(* IEC 61131-3 sources: Industry-PLC-LLM/data/PLCBEAD_repo/PLCBEAD_PLCEmbed-main/PLC-BEAD/Source/OpenPLCv2 (part 7) *)

(* ---- MB_SERVER.ST ---- *)
TYPE
	oscat_IP_FIFO128_DATA  : ARRAY [1..128] OF BYTE;
	oscat_Mailbox  : ARRAY [1..16] OF BYTE;

	oscat_NW_BUF_SHORT : ARRAY [0..1407] OF BYTE;
	oscat_NW_BUF_LONG  : ARRAY [0..4095] OF BYTE;

	oscat_IP_FIFO_DATA :
	STRUCT
		X       : oscat_IP_FIFO128_DATA; (* IP_ID FIFO Speicher          *)
		Y       : oscat_IP_FIFO128_DATA; (* IP_ID Z�hler                 *)
		ID      : BYTE;                  (* h�chste vergabene id         *)
		MAX_ID  : BYTE;                  (* maximal Anmeldungen pro ID   *)
		INIT    : BOOL;                  (* Initialisierung durchgef�hrt *)
		EMPTY   : BOOL;                  (* FIFO leer                    *)
		FULL    : BOOL;                  (* FIFO voll                    *)
		TOP     : INT;                   (* maximale anzahl in FIFO      *)
		NW      : INT;                   (* Schreibzeiger                *)
		NR      : INT;                   (* Lesezeiger                   *)
	END_STRUCT;

	oscat_IP_C:
	STRUCT
		C_MODE:			BYTE;          		(*W Mode: TCP/UCP AKTIV/PASSIV                               *)
		C_PORT:         WORD;          		(*W Portnummer                                               *)
		C_IP:           DWORD;         		(*W IP-Adresse gepackt wwxxyyzz = www.xxx.yyy.zzz            *)
		C_STATE:        BYTE;          		(*R Verbindungsstatus ON/OFF + Flanke ON/OFF                 *)
		C_ENABLE:       BOOL;          		(*W Freigabe f�r Connect                                     *)
		R_OBSERVE:      BOOL;          		(*W Empfang ueberwachen                                      *)
		TIME_RESET:     BOOL;          		(*W Alle Timer ruecksetzen                                   *)
		ERROR:          DWORD;         		(*R vvwwxxyy (vv = CON_ERROR, ww = SEN_ERROR, xx = REC_ERROR *)
		FIFO:           oscat_IP_FIFO_DATA; (*I IP FIFO Struktur                                         *)
		MAILBOX:		oscat_Mailbox;		(*I Mailbox: Datenbereich f�r Bausteindatenaustausch         *)
	END_STRUCT;

	oscat_NETWORK_BUFFER :
	STRUCT
		SIZE   : UINT;
		BUFFER : oscat_NW_BUF_LONG;
	END_STRUCT;

	oscat_NETWORK_BUFFER_SHORT :
	STRUCT
	SIZE   : UINT;
	BUFFER : oscat_NW_BUF_SHORT;
	END_STRUCT;

	oscat_aW0_255	: ARRAY [0..255] OF WORD;
	oscat_VMAP_DATA :
	STRUCT
		FC       : DWORD;
		V_ADR    : INT;
		V_SIZE   : INT;
		P_ADR    : INT;
		TIME_OUT : TIME;
	END_STRUCT;

	oscat_MB_VMAP : ARRAY [1..10] OF oscat_VMAP_DATA;

	csv_parser_demo_col : ARRAY [1..4] OF REAL;
	csv_parser_demo     : ARRAY [1..2] OF csv_parser_demo_col;

END_TYPE

FUNCTION_BLOCK MB_VMAP_Block

	VAR_IN_OUT
		VMAP :	oscat_MB_VMAP;
	END_VAR

	VAR_INPUT
		FC :	INT;
		V_ADR :	INT;
		V_CNT :	INT;
		SIZE :	INT;
	END_VAR

	VAR_OUTPUT
		P_ADR :	INT;
		P_BIT :	INT;
		ERROR :	BYTE;
	END_VAR

	VAR
		i :	INT;
		vopt :	DWORD;
		vadr :	INT;
		padr :	INT;
		mask :	DWORD;
		vsize :	INT;
		w_tmp :	WORD;
		i_tmp :	INT;
		init :	BOOL;
	END_VAR

	IF init = FALSE THEN
		init := TRUE;
		IF VMAP[1].FC = DWORD#0 THEN
			VMAP[1].FC := DWORD#16#FFFF_FFFF;
			VMAP[1].V_ADR := 0;
			VMAP[1].V_SIZE := 256;
			VMAP[1].P_ADR := 0;
		END_IF;
	END_IF;

	ERROR := BYTE#02;
	mask := SHL(DWORD#1,FC);

	IF (mask AND DWORD#2#00000000_01000000_00000000_01100000) <> DWORD#0 THEN
		V_CNT := 1;
	ELSIF V_CNT = 0 THEN
		RETURN;
	END_IF;

	FOR i := 1 TO 10 DO
		vopt := VMAP[i].FC;
		IF (vopt AND mask) <> DWORD#0 THEN
			vadr := VMAP[i].V_ADR;
			vsize := VMAP[i].V_SIZE;
			padr := VMAP[i].P_ADR;

			IF (mask AND DWORD#2#00000000_00000000_10000000_00100110) <> DWORD#0 THEN
				i_tmp := WORD_TO_INT(SHR(INT_TO_WORD(V_ADR + V_CNT -1),4))+1;
				IF i_tmp <= SIZE AND i_tmp <= vsize THEN
					w_tmp := INT_TO_WORD(V_ADR);
					P_ADR := WORD_TO_INT(SHR(w_tmp,4)) + padr;
					P_BIT := WORD_TO_INT(w_tmp AND WORD#16#000F);
					ERROR := BYTE#0;
					EXIT;
				END_IF;
			ELSIF (mask AND DWORD#2#00000000_11000001_00000000_01011000) <> DWORD#0 THEN
				IF V_ADR >= vadr AND V_ADR + V_CNT <= vadr + vsize THEN
					P_ADR := V_ADR - vadr + padr;
					IF P_ADR + V_CNT <= SIZE THEN
						ERROR := BYTE#0;
						EXIT;
					END_IF;
				END_IF;
			ELSE
				ERROR := BYTE#01;
				RETURN;
			END_IF;
		END_IF;
	END_FOR;

	IF ERROR = BYTE#0 THEN
		IF (mask AND DWORD#2#00000000_11000001_10000000_01100000) <> DWORD#0 THEN
			VMAP[i].TIME_OUT := T#1ms;
		END_IF;
	END_IF;

END_FUNCTION_BLOCK

FUNCTION _BYTE_TO_INT:INT
	VAR_INPUT
		IN :	BYTE;
	END_VAR

	_BYTE_TO_INT := USINT_TO_INT(BYTE_TO_USINT(IN));
END_FUNCTION

FUNCTION_BLOCK IP_FIFO_Block

  VAR_IN_OUT
    FIFO :	oscat_IP_FIFO_DATA;
    ID :	BYTE;
    STATE :	BYTE;
  END_VAR

  VAR
    tmp :	INT;
  END_VAR

  IF NOT FIFO.INIT THEN
    FIFO.INIT		:= TRUE;
    FIFO.NW		:= 1;
    FIFO.NR		:= 1;
    FIFO.EMPTY	:= TRUE;
    FIFO.FULL		:= FALSE;
    FIFO.TOP		:= 128;
    FIFO.MAX_ID	:= BYTE#1;
  END_IF;

  IF ID = BYTE#00 THEN
    IF FIFO.ID < INT_TO_BYTE(FIFO.TOP) THEN
      ID := USINT_TO_BYTE(BYTE_TO_USINT(FIFO.ID) + USINT#1);
      FIFO.ID := ID ;

    ELSIF STATE < BYTE#200 THEN
      STATE := BYTE#255;
    RETURN;
    END_IF;
  END_IF;

  IF STATE = BYTE#1 AND NOT FIFO.FULL THEN
    tmp := _BYTE_TO_INT(ID);
    IF FIFO.Y[tmp] < FIFO.MAX_ID THEN
      FIFO.Y[tmp] := USINT_TO_BYTE(BYTE_TO_USINT(FIFO.Y[tmp]) + USINT#1);
      tmp := FIFO.NW;
      FIFO.X[tmp] := ID;
      IF FIFO.NW = FIFO.TOP THEN FIFO.NW := 1; ELSE FIFO.NW := FIFO.NW + 1; END_IF;
      FIFO.FULL := FIFO.NW = FIFO.NR;
    FIFO.EMPTY := FALSE;
      STATE := BYTE#2;
    END_IF;
  END_IF;

  IF STATE = BYTE#2 AND NOT FIFO.EMPTY THEN
    tmp := FIFO.NR;
    IF ID = FIFO.X[tmp] THEN
      STATE := BYTE#3;
    END_IF;
  END_IF;

  IF STATE = BYTE#4 AND NOT FIFO.EMPTY THEN

    tmp := FIFO.NR;
    IF ID = FIFO.X[tmp] THEN
      tmp := _BYTE_TO_INT(ID);
      FIFO.Y[tmp] := USINT_TO_BYTE(BYTE_TO_USINT(FIFO.Y[tmp]) - USINT#1);

      IF FIFO.NR = FIFO.TOP THEN FIFO.NR := 1; ELSE FIFO.NR := FIFO.NR + 1; END_IF;
      FIFO.EMPTY := FIFO.NR = FIFO.NW;
    FIFO.FULL := FALSE;
    END_IF;
    STATE := BYTE#5;
  END_IF;

END_FUNCTION_BLOCK

FUNCTION _UDINT_TO_TIME:TIME

	VAR_INPUT
		IN :	UDINT;
	END_VAR

	_UDINT_TO_TIME := DINT_TO_TIME(UDINT_TO_DINT(IN));

END_FUNCTION

FUNCTION_BLOCK T_PLC_MS_block

	VAR_OUTPUT
		T_PLC_MS :	UDINT;
	END_VAR

	VAR_EXTERNAL
		PLC_TICKS_PER_SEC :	INT;
		PLC_SYS_TICK_CNT :	DINT;
	END_VAR

	VAR
		debug :	BOOL;(*Debug-Mode ON / OFF*)
		N :	INT;(*Debug-Faktor*)
		Offset :	UDINT;(*Debug-Offset*)
		temp :	DWORD := DWORD#1;(*Debug-Offset*)
		mode :	BOOL;(*modus*)
		faktor :	UDINT;(*Systemtakt-Faktor*)
		init :	BOOL;
		v_plc_ticks_per_sec :	UDINT;
		base :	UDINT := UDINT#1000;
	END_VAR

	IF init = FALSE THEN
		v_plc_ticks_per_sec := INT_TO_UDINT(PLC_TICKS_PER_SEC);
		IF v_plc_ticks_per_sec = UDINT#1024 THEN
			faktor := UDINT#1;
			mode := FALSE;
		ELSIF v_plc_ticks_per_sec > UDINT#0 THEN
			IF v_plc_ticks_per_sec <= base THEN
				faktor := base / v_plc_ticks_per_sec;
				mode := FALSE;
			ELSE
				faktor := v_plc_ticks_per_sec / base;
				mode := TRUE;
			END_IF;
		ELSE
			faktor := UDINT#1;
		END_IF;
		init := TRUE;
	END_IF;

	IF mode THEN
		T_PLC_MS := DINT_TO_UDINT(PLC_SYS_TICK_CNT) / faktor;
	ELSE
		T_PLC_MS := DINT_TO_UDINT(PLC_SYS_TICK_CNT) * faktor;
	END_IF;

	IF debug THEN
		T_PLC_MS := (DWORD_TO_UDINT(SHL(UDINT_TO_DWORD(T_PLC_MS),N) OR SHL(temp,N)) - UDINT#1) + Offset;
	END_IF;

END_FUNCTION_BLOCK

FUNCTION WORD_OF_BYTE:WORD
	VAR_INPUT
		B1 :	BYTE;
		B0 :	BYTE;
	END_VAR
	WORD_OF_BYTE := SHL(BYTE_TO_WORD(B1),8) OR BYTE_TO_WORD(B0);
END_FUNCTION

FUNCTION BIT_LOAD_W:WORD
	VAR_INPUT
		IN :	WORD;
		VAL :	BOOL;
		POS :	INT;
	END_VAR

	IF VAL THEN
		BIT_LOAD_W := in OR SHL(WORD#1,pos);
	ELSE
		BIT_LOAD_W := in AND (NOT SHL(WORD#1,pos));
	END_IF;
END_FUNCTION

FUNCTION_BLOCK MB_SERVER_Block

	VAR_IN_OUT
		IP_C :	oscat_IP_C;
		S_BUF :	oscat_NETWORK_BUFFER_SHORT;
		R_BUF :	oscat_NETWORK_BUFFER_SHORT;
		VMAP :	oscat_MB_VMAP;
		DATA :	oscat_aW0_255;
	END_VAR

	VAR_INPUT
		DATA_SIZE :	INT;
		ENABLE :	BOOL;
		UDP :	BOOL;
	END_VAR

	VAR_OUTPUT
		ERROR :	DWORD;
	END_VAR

	VAR
		MB_VMAP :	MB_VMAP_Block;
		adr1 :	INT;
		adr2 :	INT;
		points :	INT;
		points2 :	INT;
		coils :	BYTE;
		mask :	BYTE;
		idx1 :	INT;
		idx2 :	INT;
		bit_pos :	INT;
		count :	INT;
		fc :	INT;
		i :	INT;
		state :	INT;
		IP_STATE :	BYTE;
		IP_ID :	BYTE;
		IP_FIFO :	IP_FIFO_Block;
		w_tmp :	WORD;
		last_cycle :	TIME;
		tx :	TIME;
		T_PLC_MS :	T_PLC_MS_Block;
		t :	TON;
		ip_error :	BOOL;
	END_VAR

	T_PLC_MS();
	tx := UDINT_TO_TIME(T_PLC_MS.T_PLC_MS);

	FOR i := 1 TO 10 DO
		IF VMAP[i].TIME_OUT > T#0s THEN
			VMAP[i].TIME_OUT := VMAP[i].TIME_OUT + tx - last_cycle;
		END_IF;
	END_FOR;
	last_cycle := tx;
	ip_error := IP_C.ERROR > DWORD#0;

	CASE state OF

	00:
		IF ENABLE THEN
			state := 10;
			IP_STATE := BYTE#1;
		END_IF;

	10:
		IF IP_STATE = BYTE#3 THEN

			IP_C.C_PORT     := WORD#0;
			IP_C.C_IP       := DWORD#0;
			IP_C.C_MODE     := SEL(UDP,BYTE#4,BYTE#5);
			IP_C.TIME_RESET := TRUE;
			IP_C.C_ENABLE   := TRUE;
			IP_C.R_OBSERVE  := FALSE;
			state := 20;
		END_IF;

	20:	IF NOT ip_error THEN
			IF S_BUF.SIZE = UINT#0 AND R_BUF.SIZE > UINT#6 THEN
				IF  R_BUF.SIZE = WORD_TO_UINT(WORD_OF_BYTE(R_BUF.BUFFER[4],R_BUF.BUFFER[5])) + UINT#6 THEN
					ERROR := DWORD#00;

					FOR i := 0 TO 13 DO
						S_BUF.BUFFER[i] := R_BUF.BUFFER[i];
					END_FOR;

					fc := _BYTE_TO_INT(R_BUF.BUFFER[7]);

					adr1 := WORD_TO_INT(WORD_OF_BYTE(R_BUF.BUFFER[8],R_BUF.BUFFER[9]));
					points := WORD_TO_INT(WORD_OF_BYTE(R_BUF.BUFFER[10],R_BUF.BUFFER[11]));

					MB_VMAP(VMAP:=VMAP,FC:=fc,V_ADR:=adr1,V_CNT:=points,SIZE:=DATA_SIZE);
					VMAP:=MB_VMAP.VMAP;
					adr1:=MB_VMAP.P_ADR;
					bit_pos:=MB_VMAP.P_BIT;
					ERROR:=BYTE_TO_DWORD(MB_VMAP.ERROR);

					IF ERROR = DWORD#0 THEN
						CASE fc OF

						1..2 :
							count := 9;
							coils := BYTE#0;
							mask := BYTE#1;
							FOR i := 1 TO points DO
								IF mask = BYTE#0 THEN
									mask := BYTE#1;
									S_BUF.BUFFER[count] := coils;
									coils := BYTE#0;
									count := count + 1;
								END_IF;
								IF (DATA[adr1] AND SHL(WORD#1,bit_pos)) > WORD#0 THEN
									coils := coils OR mask;
								END_IF;

								bit_Pos := bit_Pos + 1;
								IF bit_pos > 15 THEN
									adr1 := adr1 + 1;
									bit_pos := 0;
								END_IF;

								mask := SHL(mask,1);
							END_FOR;
							S_BUF.BUFFER[Count] := coils;

							S_BUF.BUFFER[8] := INT_TO_BYTE(count - 8);
							S_BUF.SIZE := INT_TO_UINT(count + 1);

						3..4 :
							idx1 := 07;
							count := adr1 + points - 1;
							FOR i := adr1 TO count DO
								idx1 := idx1 + 2;
								idx2 := idx1 + 1;
								w_tmp := DATA[i];
								S_BUF.BUFFER[idx1] := WORD_TO_BYTE(SHR(w_tmp,8));
								S_BUF.BUFFER[idx2] := WORD_TO_BYTE(w_tmp);
							END_FOR;
							S_BUF.BUFFER[8] := SHL(INT_TO_BYTE(points),1);
							S_BUF.SIZE := INT_TO_UINT(idx2 + 1);
						5 :
							DATA[adr1]:=BIT_LOAD_W(DATA[adr1],R_BUF.BUFFER[10]>BYTE#0,bit_pos);
							S_BUF.SIZE := UINT#12;
						6 :
							DATA[adr1] := WORD_OF_BYTE(R_BUF.BUFFER[10],R_BUF.BUFFER[11]);
							S_BUF.SIZE := UINT#12;
						15 :
							mask := BYTE#1;
							idx1 := 13;
							FOR i := 1 TO points DO
								DATA[adr1]:=BIT_LOAD_W(DATA[adr1],(R_BUF.BUFFER[idx1] AND mask)>BYTE#0,bit_pos);
								bit_pos := bit_pos + 1;
								IF bit_pos > 15 THEN
									adr1 := adr1 + 1;
									bit_pos := 0;
								END_IF;
								mask := ROL(mask,1);
								IF mask = BYTE#1 THEN
									idx1 := idx1 +1;
								END_IF;
							END_FOR;
							S_BUF.SIZE := UINT#12;
						16 :
							idx1 := 11;
							count := adr1 + points -1;
							FOR i := adr1 TO Count DO
								idx1 := idx1 + 2;
								idx2 := idx1 + 1;
								Data[i] := WORD_OF_BYTE(R_BUF.BUFFER[idx1],R_BUF.BUFFER[idx2]);
							END_FOR;
							S_BUF.SIZE := UINT#12;
						22 :
							w_tmp := WORD_OF_BYTE(R_BUF.BUFFER[11],R_BUF.BUFFER[11]);
							DATA[adr1] := (DATA[adr1] AND w_tmp) OR (WORD_OF_BYTE(R_BUF.BUFFER[12],R_BUF.BUFFER[13]) AND (NOT w_tmp));
							S_BUF.SIZE := UINT#14;
						23 :
							adr2 := WORD_TO_INT(WORD_OF_BYTE(R_BUF.BUFFER[12],R_BUF.BUFFER[13]));
							points2 := WORD_TO_INT(WORD_OF_BYTE(R_BUF.BUFFER[14],R_BUF.BUFFER[15]));

							MB_VMAP(VMAP:=VMAP,FC:=16,V_ADR:=adr2,V_CNT:=points2,SIZE:=DATA_SIZE);
							VMAP:=MB_VMAP.VMAP;
							adr2:=MB_VMAP.P_ADR;
							ERROR:=BYTE_TO_DWORD(MB_VMAP.ERROR);

							IF ERROR = DWORD#0 THEN
								idx1 := 15;
								count := adr2 + points2 -1;
								FOR i := adr2 TO count DO
									idx1 := idx1 + 2;
									idx2 := idx1 + 1;
									Data[i] := WORD_OF_BYTE(R_BUF.BUFFER[idx1],R_BUF.BUFFER[idx2]);
								END_FOR;

								idx1 := 07;
								count := adr1 + points - 1;
								FOR i := adr1 TO count DO
									idx1 := idx1 + 2;
									idx2 := idx1 + 1;
									w_tmp := DATA[i];
									S_BUF.BUFFER[idx1] := WORD_TO_BYTE(SHR(w_tmp,8));
									S_BUF.BUFFER[idx2] := WORD_TO_BYTE(w_tmp);
								END_FOR;
								S_BUF.BUFFER[8] := SHL(INT_TO_BYTE(points),1);
								S_BUF.SIZE := INT_TO_UINT(idx2 + 1);

							END_IF;

						ELSE
							ERROR := DWORD#01;
						END_CASE;
					END_IF;
				END_IF;

				IF ERROR > DWORD#0 THEN
					S_BUF.BUFFER[7] := S_BUF.BUFFER[7] OR BYTE#2#1000_0000;
					S_BUF.BUFFER[8] := DWORD_TO_BYTE(ERROR);
					S_BUF.SIZE := UINT#9;
				END_IF;

				S_BUF.BUFFER[4] := BYTE#0;
				S_BUF.BUFFER[5] := UINT_TO_BYTE(S_BUF.SIZE - UINT#6);

			END_IF;
		ELSE
			ERROR := IP_C.ERROR;
		END_IF;

		t(IN:= ip_error, PT:=T#5s);
		IF t.Q THEN
			IP_C.TIME_RESET := TRUE;
		END_IF;

		R_BUF.SIZE := UINT#0;

		IF ENABLE = FALSE THEN
			IP_STATE := BYTE#4;
			state := 00;
		END_IF;
	END_CASE;

	IP_FIFO(FIFO:=IP_C.FIFO,STATE:=IP_STATE,ID:=IP_ID);
	IP_C.FIFO:=IP_FIFO.FIFO;
	IP_STATE := IP_FIFO.STATE;
	IP_ID:=IP_FIFO.ID;

END_FUNCTION_BLOCK

PROGRAM program0
	VAR
		IP_C :	oscat_IP_C;
		S_BUF :	oscat_NETWORK_BUFFER_SHORT;
		R_BUF :	oscat_NETWORK_BUFFER_SHORT;
		VMAP :	oscat_MB_VMAP;
		DATA :	oscat_aW0_255;
		DATA_SIZE :	INT;
		ENABLE :	BOOL;
		UDP :	BOOL;
		ERROR :	DWORD;

		func_block : MB_SERVER_Block;
	END_VAR
	func_block.IP_C := IP_C;
	func_block.S_BUF := S_BUF;
	func_block.R_BUF := R_BUF;
	func_block.VMAP := VMAP;
	func_block.DATA := DATA;
	func_block.DATA_SIZE := DATA_SIZE;
	func_block.ENABLE := ENABLE;
	func_block.UDP := UDP;

	func_block();
  	IP_C  := func_block.IP_C;
	S_BUF  := func_block.S_BUF;
	R_BUF  := func_block.R_BUF;
	VMAP  := func_block.VMAP;
	DATA  := func_block.DATA;
	ERROR  := func_block.ERROR;

END_PROGRAM

CONFIGURATION Config0

	VAR_GLOBAL
		PLC_TICKS_PER_SEC :	INT;
		PLC_SYS_TICK_CNT :	DINT;
	END_VAR

  	RESOURCE Res0 ON PLC
    	TASK task0(INTERVAL := T#20ms,PRIORITY := 0);
    	PROGRAM instance0 WITH task0 : program0;
  	END_RESOURCE

END_CONFIGURATION

(* ---- MB_VMAP.ST ---- *)
TYPE
  oscat_VMAP_DATA :
  STRUCT
	FC       : DWORD;
    V_ADR    : INT;
    V_SIZE   : INT;
    P_ADR    : INT;
	TIME_OUT : TIME;
  END_STRUCT;

  oscat_MB_VMAP : ARRAY [1..10] OF oscat_VMAP_DATA;

  csv_parser_demo_col : ARRAY [1..4] OF REAL;
  csv_parser_demo     : ARRAY [1..2] OF csv_parser_demo_col;

END_TYPE

FUNCTION_BLOCK MB_VMAP_Block

	VAR_IN_OUT
		VMAP :	oscat_MB_VMAP;
	END_VAR

	VAR_INPUT
		FC :	INT;
		V_ADR :	INT;
		V_CNT :	INT;
		SIZE :	INT;
	END_VAR

	VAR_OUTPUT
		P_ADR :	INT;
		P_BIT :	INT;
		ERROR :	BYTE;
	END_VAR

	VAR
		i :	INT;
		vopt :	DWORD;
		vadr :	INT;
		padr :	INT;
		mask :	DWORD;
		vsize :	INT;
		w_tmp :	WORD;
		i_tmp :	INT;
		init :	BOOL;
	END_VAR

	IF init = FALSE THEN
		init := TRUE;
		IF VMAP[1].FC = DWORD#0 THEN
			VMAP[1].FC := DWORD#16#FFFF_FFFF;
			VMAP[1].V_ADR := 0;
			VMAP[1].V_SIZE := 256;
			VMAP[1].P_ADR := 0;
		END_IF;
	END_IF;

	ERROR := BYTE#02;
	mask := SHL(DWORD#1,FC);

	IF (mask AND DWORD#2#00000000_01000000_00000000_01100000) <> DWORD#0 THEN
		V_CNT := 1;
	ELSIF V_CNT = 0 THEN
		RETURN;
	END_IF;

	FOR i := 1 TO 10 DO
		vopt := VMAP[i].FC;
		IF (vopt AND mask) <> DWORD#0 THEN
			vadr := VMAP[i].V_ADR;
			vsize := VMAP[i].V_SIZE;
			padr := VMAP[i].P_ADR;

			IF (mask AND DWORD#2#00000000_00000000_10000000_00100110) <> DWORD#0 THEN
				i_tmp := WORD_TO_INT(SHR(INT_TO_WORD(V_ADR + V_CNT -1),4))+1;
				IF i_tmp <= SIZE AND i_tmp <= vsize THEN
					w_tmp := INT_TO_WORD(V_ADR);
					P_ADR := WORD_TO_INT(SHR(w_tmp,4)) + padr;
					P_BIT := WORD_TO_INT(w_tmp AND WORD#16#000F);
					ERROR := BYTE#0;
					EXIT;
				END_IF;
			ELSIF (mask AND DWORD#2#00000000_11000001_00000000_01011000) <> DWORD#0 THEN
				IF V_ADR >= vadr AND V_ADR + V_CNT <= vadr + vsize THEN
					P_ADR := V_ADR - vadr + padr;
					IF P_ADR + V_CNT <= SIZE THEN
						ERROR := BYTE#0;
						EXIT;
					END_IF;
				END_IF;
			ELSE
				ERROR := BYTE#01;
				RETURN;
			END_IF;
		END_IF;
	END_FOR;

	IF ERROR = BYTE#0 THEN
		IF (mask AND DWORD#2#00000000_11000001_10000000_01100000) <> DWORD#0 THEN
			VMAP[i].TIME_OUT := T#1ms;
		END_IF;
	END_IF;

END_FUNCTION_BLOCK

PROGRAM program0
	VAR
		VMAP :	oscat_MB_VMAP;
		FC :	INT;
		V_ADR :	INT;
		V_CNT :	INT;
		SIZE :	INT;
		P_ADR :	INT;
		P_BIT :	INT;
		ERROR :	BYTE;

		func_block : MB_VMAP_Block;
	END_VAR
	func_block.VMAP := VMAP;
	func_block.V_ADR := V_ADR;
	func_block.FC := FC;
	func_block.V_CNT := V_CNT;
	func_block.SIZE := SIZE;

	func_block();
  	VMAP  := func_block.VMAP;
	P_ADR  := func_block.P_ADR;
	P_BIT  := func_block.P_BIT;
	ERROR  := func_block.ERROR;
END_PROGRAM

CONFIGURATION Config0
	RESOURCE Res0 ON PLC
		TASK task0(INTERVAL := T#20ms,PRIORITY := 0);
		PROGRAM instance0 WITH task0 : program0;
	END_RESOURCE
END_CONFIGURATION

(* ---- MESSAGE_4R.ST ---- *)
FUNCTION INC1:INT

	VAR_INPUT
		X :	INT;
		N :	INT;
	END_VAR

	IF X >= N - 1 THEN
		INC1 := 0;
	ELSE
		INC1 := X + 1;
	END_IF;
END_FUNCTION

FUNCTION_BLOCK MESSAGE_4R_Block

	VAR_INPUT
		M0 :	STRING;
		M1 :	STRING;
		M2 :	STRING;
		M3 :	STRING;
		MM :	INT := 3;
		ENQ :	BOOL := TRUE;
		CLK :	BOOL := TRUE;
		T1 :	TIME := T#3s;
	END_VAR

	VAR_OUTPUT
		MX :	STRING;
		MN :	INT;
		TR :	BOOL;
	END_VAR

	VAR
		timer :	TON;
		edge :	BOOL;
	END_VAR

	TR := FALSE;
	IF ENQ THEN
		IF (NOT edge AND clk) OR timer.q THEN
				MN := INC1(MN, MM);
				TR := TRUE;
				timer(in := FALSE);
				CASE MN OF
					0 : MX := M0;
					1 : MX := M1;
					2 : MX := M2;
					3 : MX := M3;
				END_CASE;
		END_IF;
		edge := clk;
		timer( in := CLK, pt := T1);
	ELSE
		MX := '';
		MN := 0;
	END_IF;

END_FUNCTION_BLOCK

PROGRAM program0

	VAR
		M0 :	STRING;
		M1 :	STRING;
		M2 :	STRING;
		M3 :	STRING;
		MM :	INT;
		ENQ :	BOOL;
		CLK :	BOOL;
		T1 :	TIME;

		MX :	STRING;
		MN :	INT;
		TR :	BOOL;

		func_block : MESSAGE_4R_Block;
	END_VAR

	func_block.M0 := M0;
	func_block.M1 := M1;
	func_block.M2 := M2;
	func_block.M3 := M3;
	func_block.MM := MM;
	func_block.ENQ := ENQ;
	func_block.CLK := CLK;
	func_block.T1 := T1;

	func_block();

	MX := func_block.MX;
	MN := func_block.MN;
	TR := func_block.TR;

END_PROGRAM

CONFIGURATION Config0

	RESOURCE Res0 ON PLC
		TASK task0(INTERVAL := T#20ms,PRIORITY := 0);
		PROGRAM instance0 WITH task0 : program0;
	END_RESOURCE

END_CONFIGURATION

(* ---- MESSAGE_8.ST ---- *)
FUNCTION_BLOCK MESSAGE_8_Block

	VAR_INPUT
		IN1 :	BOOL;
		IN2 :	BOOL;
		IN3 :	BOOL;
		IN4 :	BOOL;
		IN5 :	BOOL;
		IN6 :	BOOL;
		IN7 :	BOOL;
		IN8 :	BOOL;
		S1 :	STRING;
		S2 :	STRING;
		S3 :	STRING;
		S4 :	STRING;
		S5 :	STRING;
		S6 :	STRING;
		S7 :	STRING;
		S8 :	STRING;
	END_VAR

	VAR_OUTPUT
		M :	STRING;
	END_VAR

	IF in1 THEN
		M := S1;
	ELSIF in2 THEN
		M := S2;
	ELSIF in3 THEN
		M := S3;
	ELSIF in4 THEN
		M := S4;
	ELSIF in5 THEN
		M := S5;
	ELSIF in6 THEN
		M := S6;
	ELSIF in7 THEN
		M := S7;
	ELSIF in8 THEN
		M := S8;
	ELSE
		M := '';
	END_IF;

END_FUNCTION_BLOCK

PROGRAM program0

	VAR
		IN1 :	BOOL;
		IN2 :	BOOL;
		IN3 :	BOOL;
		IN4 :	BOOL;
		IN5 :	BOOL;
		IN6 :	BOOL;
		IN7 :	BOOL;
		IN8 :	BOOL;
		S1 :	STRING;
		S2 :	STRING;
		S3 :	STRING;
		S4 :	STRING;
		S5 :	STRING;
		S6 :	STRING;
		S7 :	STRING;
		S8 :	STRING;

		M :	STRING;

		func_block : MESSAGE_8_Block;
	END_VAR

	func_block.IN1 := IN1;
	func_block.IN2 := IN2;
	func_block.IN3 := IN3;
	func_block.IN4 := IN4;
	func_block.IN5 := IN5;
	func_block.IN6 := IN6;
	func_block.IN7 := IN7;
	func_block.IN8 := IN8;
	func_block.S1 := S1;
	func_block.S2 := S2;
	func_block.S3 := S3;
	func_block.S4 := S4;
	func_block.S5 := S5;
	func_block.S6 := S6;
	func_block.S7 := S7;
	func_block.S8 := S8;

	func_block();

	M  := func_block.M;

END_PROGRAM

CONFIGURATION Config0

	VAR_GLOBAL
		PLC_TICKS_PER_SEC :	INT;
		PLC_SYS_TICK_CNT :	DINT;
	END_VAR

	RESOURCE Res0 ON PLC
		TASK task0(INTERVAL := T#20ms,PRIORITY := 0);
		PROGRAM instance0 WITH task0 : program0;
	END_RESOURCE

END_CONFIGURATION

(* ---- METER.ST ---- *)
TYPE REAL2:

	STRUCT
		R1 : REAL;
		RX : REAL;
	END_STRUCT;

END_TYPE

FUNCTION_BLOCK R2_ADD_Block

	VAR_INPUT
		X :	REAL2;
		Y :	REAL;
	END_VAR

	VAR_OUTPUT
		R2_ADD :	REAL2;
	END_VAR

	VAR
		temp :	REAL;
	END_VAR

	temp := X.RX;
	R2_ADD.RX := Y + X.R1 + X.RX;
	R2_ADD.R1 := temp - R2_ADD.RX + Y + X.R1;

END_FUNCTION_BLOCK

FUNCTION_BLOCK T_PLC_MS_Block
	VAR_OUTPUT
		T_PLC_MS :	UDINT;
	END_VAR

	VAR_EXTERNAL
		PLC_TICKS_PER_SEC :	INT;
		PLC_SYS_TICK_CNT :	DINT;
	END_VAR

	VAR
		debug :	BOOL;(*Debug-Mode ON / OFF*)
		N :	INT;(*Debug-Faktor*)
		Offset :	UDINT;(*Debug-Offset*)
		temp :	DWORD := DWORD#1;(*Debug-Offset*)
		mode :	BOOL;(*modus*)
		faktor :	UDINT;(*Systemtakt-Faktor*)
		init :	BOOL;
		v_plc_ticks_per_sec :	UDINT;
		base :	UDINT := UDINT#1000;
	END_VAR

	IF init = FALSE THEN
		v_plc_ticks_per_sec := INT_TO_UDINT(PLC_TICKS_PER_SEC);
		IF v_plc_ticks_per_sec = UDINT#1024 THEN
			faktor := UDINT#1;
			mode := FALSE;
		ELSIF v_plc_ticks_per_sec > UDINT#0 THEN
			IF v_plc_ticks_per_sec <= base THEN
				faktor := base / v_plc_ticks_per_sec;
				mode := FALSE;
			ELSE
				faktor := v_plc_ticks_per_sec / base;
				mode := TRUE;
			END_IF;
		ELSE
			faktor := UDINT#1;
		END_IF;
		init := TRUE;
	END_IF;

	IF mode THEN
		T_PLC_MS := DINT_TO_UDINT(PLC_SYS_TICK_CNT) / faktor;
	ELSE
		T_PLC_MS := DINT_TO_UDINT(PLC_SYS_TICK_CNT) * faktor;
	END_IF;

	IF debug THEN
		T_PLC_MS := (DWORD_TO_UDINT(SHL(UDINT_TO_DWORD(T_PLC_MS),N) OR SHL(temp,N)) - UDINT#1) + Offset;
	END_IF;
END_FUNCTION_BLOCK

FUNCTION_BLOCK METER_Block

	VAR_INPUT
		M1 :	REAL;
		M2 :	REAL;
		I1 :	BOOL;
		I2 :	BOOL;
		D :	REAL := 1.0;
		RST :	BOOL;
	END_VAR

	VAR_IN_OUT
		MX :	REAL;
	END_VAR

	VAR RETAIN
		MR :	REAL2;
	END_VAR

	VAR
		MX1 :	REAL;(*current consumption value on M1 and M2*)
		MX2 :	REAL;(*current consumption value on M1 and M2*)
		tx :	UDINT;
		last :	UDINT;
		tc :	REAL;
		init :	BOOL;
		T_PLC_MS :	T_PLC_MS_Block;
		R2_ADD :	R2_ADD_Block;
	END_VAR

	T_PLC_MS();
	tx:= T_PLC_MS.T_PLC_MS;
	IF NOT init THEN
		init := TRUE;
		last := tx;
		mr.RX := mx;
		mr.R1 := 0.0;
	ELSIF tx = last THEN
		RETURN;
	ELSE
		tc := UDINT_TO_REAL(tx - last) * 0.001;
	END_IF;
	last := tx;

	(* reset *)
	IF rst THEN
		mr.R1 := 0.0;
		mr.RX := 0.0;
	ELSE
		MX1 := SEL(I1,0.0,M1);
		MX2 := SEL(I2,0.0,M2);
		R2_ADD(X:=MR,Y:=(SEL(I1,0.0,mx1) + SEL(I2, 0.0, mx2)) / D * TC);
		MR:=R2_ADD.R2_ADD;
		MX := mr.RX;
	END_IF;

END_FUNCTION_BLOCK

PROGRAM program0

	VAR
		M1 :	REAL;
		M2 :	REAL;
		I1 :	BOOL;
		I2 :	BOOL;
		D :	REAL := 1.0;
		RST :	BOOL;

		MX :	REAL;

		func_block : METER_Block;
	END_VAR

	func_block.M1 := M1;
	func_block.M2 := M2;
	func_block.I1 := I1;
	func_block.I2 := I2;
	func_block.D := D;
	func_block.RST := RST;
	func_block.MX := MX;

	func_block();

	MX  := func_block.MX;

END_PROGRAM

CONFIGURATION Config0

	VAR_GLOBAL
		PLC_TICKS_PER_SEC :	INT;
		PLC_SYS_TICK_CNT :	DINT;
	END_VAR

	RESOURCE Res0 ON PLC
		TASK task0(INTERVAL := T#20ms,PRIORITY := 0);
		PROGRAM instance0 WITH task0 : program0;
	END_RESOURCE

END_CONFIGURATION

(* ---- METER_STAT.ST ---- *)
FUNCTION DAY_OF_WEEK:INT

	VAR_INPUT
		IDATE :	UDINT;
	END_VAR

	DAY_OF_WEEK := UDINT_TO_INT((idate / UDINT#86400 + UDINT#3) MOD UDINT#7) + INT#01;
END_FUNCTION

FUNCTION LEAP_OF_DATE:BOOL

	VAR_INPUT
		IDATE :	UDINT;
	END_VAR

	LEAP_OF_DATE := SHL(UDINT_TO_DWORD((idate + UDINT#43200) / UDINT#31557600), 30) = DWORD#16#80000000;
END_FUNCTION

FUNCTION DAY_OF_YEAR:INT
	VAR_INPUT
		IDATE :	UDINT;
	END_VAR

	DAY_OF_YEAR := UDINT_TO_INT(((idate) / UDINT#86400) MOD UDINT#1461);
	IF DAY_OF_YEAR > 729 THEN
		IF DAY_OF_YEAR > 1095 THEN DAY_OF_YEAR := DAY_OF_YEAR - 1095; ELSE DAY_OF_YEAR := DAY_OF_YEAR - 729; END_IF;
	ELSIF DAY_OF_YEAR > 364 THEN
		DAY_OF_YEAR := DAY_OF_YEAR - 364;
	ELSE
		DAY_OF_YEAR := DAY_OF_YEAR + 1;
	END_IF;
END_FUNCTION

FUNCTION MONTH_OF_DATE:INT

	VAR_INPUT
		IDATE :	UDINT;
	END_VAR

	MONTH_OF_DATE := DAY_OF_YEAR(idate);
	IF MONTH_OF_DATE < 32 THEN
		MONTH_OF_DATE := 1;
	ELSIF LEAP_OF_DATE((IDATE)) THEN
		MONTH_OF_DATE := (MONTH_OF_DATE * 53 + 1668) / 1623;
	ELSE
		MONTH_OF_DATE := (MONTH_OF_DATE * 53 + 1700) / 1620;
	END_IF;
END_FUNCTION

FUNCTION YEAR_OF_DATE:INT
	VAR_INPUT
		IDATE :	UDINT;
	END_VAR

	YEAR_OF_DATE := UDINT_TO_INT((idate+UDINT#43200) / UDINT#31557600 + UDINT#1970);
END_FUNCTION

FUNCTION_BLOCK METER_STAT_Block

	VAR_INPUT
		IN :	REAL;
		DI :	UDINT;
		RST :	BOOL;
	END_VAR

	VAR_IN_OUT
		LAST_DAY :	REAL;
		CURRENT_DAY :	REAL;
		LAST_WEEK :	REAL;
		CURRENT_WEEK :	REAL;
		LAST_MONTH :	REAL;
		CURRENT_MONTH :	REAL;
		LAST_YEAR :	REAL;
		CURRENT_YEAR :	REAL;
	END_VAR

	VAR RETAIN
		year_start :	REAL;
		month_start :	REAL;
		week_start :	REAL;
		day_start :	REAL;
		last_run :	UDINT;
	END_VAR

	IF rst THEN
		Last_Day := 0.0;
		Current_Day := 0.0;
		Day_start := IN;
		Last_week := 0.0;
		Current_week := 0.0;
		Week_start := in;
		Last_month := 0.0;
		Current_month := 0.0;
		month_start := in;
		last_year := 0.0;
		current_year := 0.0;
		year_start := in;
	ELSE
		Current_Day := IN - Day_Start;
		Current_Week := In - Week_Start;
		Current_Month := IN - Month_Start;
		Current_Year := IN - Year_Start;
	END_IF;

	IF YEAR_OF_DATE(DI) > YEAR_OF_DATE(last_run) THEN
		(* a new year has started *)
		last_year := current_year;
		current_year := 0.0;
		year_start := in;
		last_month := current_month;
		current_month := 0.0;
		month_start := in;
		last_day := current_day;
		current_day := 0.0;
		day_start := in;
	ELSIF MONTH_OF_DATE(DI) > MONTH_OF_DATE(last_run) THEN
		(* a new month has started, january is alrerady done by year change *)
		last_month := current_month;
		current_month := 0.0;
		month_start := in;
		last_day := current_day;
		current_day := 0.0;
		day_start := in;
	ELSIF DAY_OF_YEAR(di) > DAY_OF_YEAR(last_run) THEN
		(* day has chaged, first day of year and first day of month has already been taken care of *)
		last_day := current_day;
		current_day := 0.0;
		day_start := in;
	END_IF;
	IF DAY_OF_WEEK(DI) < DAY_OF_WEEK(last_run) THEN
		(* a new week has started *)
		last_week := current_week;
		current_week := 0.0;
		week_start := in;
	END_IF;
	last_run := di;

END_FUNCTION_BLOCK

PROGRAM program0

	VAR
		IN :	REAL;
		DI :	UDINT;
		RST :	BOOL;

		LAST_DAY :	REAL;
		CURRENT_DAY :	REAL;
		LAST_WEEK :	REAL;
		CURRENT_WEEK :	REAL;
		LAST_MONTH :	REAL;
		CURRENT_MONTH :	REAL;
		LAST_YEAR :	REAL;
		CURRENT_YEAR :	REAL;

		func_block : METER_STAT_Block;
	END_VAR

	func_block.IN := IN;
	func_block.DI := DI;
	func_block.RST := RST;
	func_block.LAST_DAY := LAST_DAY;
	func_block.CURRENT_DAY := CURRENT_DAY;
	func_block.LAST_WEEK := LAST_WEEK;
	func_block.CURRENT_WEEK := CURRENT_WEEK;
	func_block.LAST_MONTH := LAST_MONTH;
	func_block.CURRENT_MONTH := CURRENT_MONTH;
	func_block.LAST_YEAR := LAST_YEAR;
	func_block.CURRENT_YEAR := CURRENT_YEAR;

	func_block();

	LAST_DAY  := func_block.LAST_DAY;
	CURRENT_DAY  := func_block.CURRENT_DAY;
	LAST_WEEK  := func_block.LAST_WEEK;
	CURRENT_WEEK  := func_block.CURRENT_WEEK;
	LAST_MONTH  := func_block.LAST_MONTH;
	CURRENT_MONTH  := func_block.CURRENT_MONTH;
	LAST_YEAR  := func_block.LAST_YEAR;
	CURRENT_YEAR  := func_block.CURRENT_YEAR;

END_PROGRAM

CONFIGURATION Config0

	VAR_GLOBAL
		PLC_TICKS_PER_SEC :	INT;
		PLC_SYS_TICK_CNT :	DINT;
	END_VAR

	RESOURCE Res0 ON PLC
		TASK task0(INTERVAL := T#20ms,PRIORITY := 0);
		PROGRAM instance0 WITH task0 : program0;
	END_RESOURCE

END_CONFIGURATION

(* ---- MIRROR.ST ---- *)
FUNCTION_BLOCK MIRROR_Block

	VAR_INPUT
		STR :	STRING;
	END_VAR

	VAR_OUTPUT
		MIRROR :	STRING;
	END_VAR

	VAR
		i :	INT;
		st_temp :	STRING;
	END_VAR

	mirror := '';
	i := LEN(str);
	WHILE i > 0 DO
	st_temp := MID(str,1,i);
	mirror := CONCAT(mirror,st_temp);
	i := i -1;
	END_WHILE;

END_FUNCTION_BLOCK

PROGRAM program0

	VAR
		STR :	STRING;
		MIRROR :	STRING;
		func_block : MIRROR_Block;
	END_VAR
	func_block.STR := STR;
	func_block();
	MIRROR  := func_block.MIRROR;

END_PROGRAM

CONFIGURATION Config0

	RESOURCE Res0 ON PLC
		TASK task0(INTERVAL := T#20ms,PRIORITY := 0);
		PROGRAM instance0 WITH task0 : program0;
	END_RESOURCE

END_CONFIGURATION

(* ---- MONTH_TO_STRING.ST ---- *)
TYPE
  oscat_ELEMENT_MONTHS 	: ARRAY [1..12] OF STRING;
  oscat_MONTHS			: ARRAY [1..3]  OF oscat_ELEMENT_MONTHS := [0, 0, 0];
  oscat_ELEMENT_MONTHS3	: ARRAY [1..12] OF STRING;
  oscat_MONTHS3			: ARRAY [1..3]  OF oscat_ELEMENT_MONTHS3 := [0,0,0];
END_TYPE

TYPE oscat_LANGUAGE:
  STRUCT
    DEFAULT 	: INT;
	LMAX    	: INT;
  END_STRUCT;
END_TYPE

FUNCTION_BLOCK SETUP_LANGUAGE_Block

	VAR_IN_OUT
		LANGUAGE :	oscat_LANGUAGE;
	END_VAR

	VAR
		init :	BOOL;
	END_VAR

	IF init THEN RETURN; END_IF;
	init := TRUE;

	LANGUAGE.DEFAULT  := 1; (* 1=english, 2=german 3=french *)
	LANGUAGE.LMAX := 3;
END_FUNCTION_BLOCK

FUNCTION_BLOCK SETUP_MONTHS3_Block

	VAR_IN_OUT
		MONTHS3 :	oscat_MONTHS3;
	END_VAR

	VAR
		init :	BOOL;
	END_VAR

	IF init THEN RETURN; END_IF;
	init := TRUE;

	(* ---- english --- *)
	MONTHS3[1][01] := 'Jan';
	MONTHS3[1][02] := 'Feb';
	MONTHS3[1][03] := 'Mar';
	MONTHS3[1][04] := 'Apr';
	MONTHS3[1][05] := 'May';
	MONTHS3[1][06] := 'Jun';
	MONTHS3[1][07] := 'Jul';
	MONTHS3[1][08] := 'Aug';
	MONTHS3[1][09] := 'Sep';
	MONTHS3[1][10] := 'Oct';
	MONTHS3[1][11] := 'Nov';
	MONTHS3[1][12] := 'Dec';

	(* ---- german --- *)
	MONTHS3[2][01] := 'Jan';
	MONTHS3[2][02] := 'Feb';
	MONTHS3[2][03] := 'Mrz';
	MONTHS3[2][04] := 'Apr';
	MONTHs3[2][05] := 'Mai';
	MONTHS3[2][06] := 'Jun';
	MONTHS3[2][07] := 'Jul';
	MONTHS3[2][08] := 'Aug';
	MONTHS3[2][09] := 'Sep';
	MONTHS3[2][10] := 'Okt';
	MONTHS3[2][11] := 'Nov';
	MONTHS3[2][12] := 'Dez';

	(* ---- french --- *)
	MONTHS3[3][01] := 'Jan';
	MONTHS3[3][02] := 'Fev';
	MONTHS3[3][03] := 'Mar';
	MONTHS3[3][04] := 'Avr';
	MONTHs3[3][05] := 'Mai';
	MONTHS3[3][06] := 'Jun';
	MONTHS3[3][07] := 'Jul';
	MONTHS3[3][08] := 'Aou';
	MONTHS3[3][09] := 'Sep';
	MONTHS3[3][10] := 'Oct';
	MONTHS3[3][11] := 'Nov';
	MONTHS3[3][12] := 'Dec';
	(*@KEY@: END_WORKSHEET *)
END_FUNCTION_BLOCK

FUNCTION_BLOCK SETUP_MONTHS_Block

	VAR_IN_OUT
		MONTHS :	oscat_MONTHS;
	END_VAR

	VAR
		init :	BOOL;
	END_VAR

	IF init THEN RETURN; END_IF;
	init := TRUE;

	(* ---- english --- *)
	MONTHS[1][01] := 'January';
	MONTHS[1][02] := 'February';
	MONTHS[1][03] := 'March';
	MONTHS[1][04] := 'April';
	MONTHS[1][05] := 'May';
	MONTHS[1][06] := 'June';
	MONTHS[1][07] := 'July';
	MONTHS[1][08] := 'August';
	MONTHS[1][09] := 'September';
	MONTHS[1][10] := 'October';
	MONTHS[1][11] := 'November';
	MONTHS[1][12] := 'December';

	(* ---- german --- *)
	MONTHS[2][01] := 'Januar';
	MONTHS[2][02] := 'Februar';
	MONTHS[2][03] := 'March';
	MONTHS[2][04] := 'April';
	MONTHS[2][05] := 'Mai';
	MONTHS[2][06] := 'Juni';
	MONTHS[2][07] := 'Juli';
	MONTHS[2][08] := 'August';
	MONTHS[2][09] := 'September';
	MONTHS[2][10] := 'Oktober';
	MONTHS[2][11] := 'November';
	MONTHS[2][12] := 'Dezember';

	(* ---- french --- *)
	MONTHS[3][01] := 'Janvier';
	MONTHS[3][02] := 'Fvrier';
	MONTHS[3][03] := 'mars';
	MONTHS[3][04] := 'Avril';
	MONTHS[3][05] := 'Mai';
	MONTHS[3][06] := 'Juin';
	MONTHS[3][07] := 'Juillet';
	MONTHS[3][08] := 'Aot';
	MONTHS[3][09] := 'Septembre';
	MONTHS[3][10] := 'Octobre';
	MONTHS[3][11] := 'Novembre';
	MONTHS[3][12] := 'Decembre';
END_FUNCTION_BLOCK

FUNCTION_BLOCK MONTH_TO_STRING_Block

	VAR_INPUT
		MTH :	INT;
		LANG :	INT;
		LX :	INT;
	END_VAR

	VAR_OUTPUT
		MONTH_TO_STRING :	STRING;
	END_VAR

	VAR
		LY :	INT;
		SETUP_MONTHS :	SETUP_MONTHS_Block;
		MONTHS :	oscat_MONTHS;
		SETUP_MONTHS3 :	SETUP_MONTHS3_Block;
		MONTHS3 :	oscat_MONTHS3;
		SETUP_LANGUAGE :	SETUP_LANGUAGE_Block;
		LANGUAGE :	oscat_LANGUAGE;
	END_VAR

	SETUP_MONTHS(MONTHS:=MONTHS);
	MONTHS:=SETUP_MONTHS.MONTHS;
	SETUP_MONTHS3(MONTHS3:=MONTHS3);
	MONTHS3:=SETUP_MONTHS3.MONTHS3;
	SETUP_LANGUAGE(LANGUAGE:=LANGUAGE);
	LANGUAGE:=SETUP_LANGUAGE.LANGUAGE;

	IF LANG = 0 THEN Ly := LANGUAGE.DEFAULT; ELSE ly := MIN(LANG, language.LMAX); END_IF;
	IF MTH < 1 OR MTH > 12 THEN
		RETURN;
	ELSIF LX = 0 THEN
		MONTH_TO_STRING := MONTHS[ly][MTH];
	ELSIF Lx = 3 THEN
		MONTH_TO_STRING := MONTHS3[ly][MTH];
	END_IF;

END_FUNCTION_BLOCK

PROGRAM program0
	VAR
		MTH :	INT;
		LANG :	INT;
		LX :	INT;
		MONTH_TO_STRING :	STRING;
		func_block : MONTH_TO_STRING_Block;
	END_VAR
		func_block.MTH  := MTH;
		func_block.LANG  := LANG;
		func_block.LX  := LX;
		func_block();
		MONTH_TO_STRING := func_block.MONTH_TO_STRING;
END_PROGRAM

CONFIGURATION Config0
	RESOURCE Res0 ON PLC
		TASK task0(INTERVAL := T#20ms,PRIORITY := 0);
		PROGRAM instance0 WITH task0 : program0;
	END_RESOURCE
END_CONFIGURATION

(* ---- MOON_PHASE.ST ---- *)
FUNCTION TIME_TO_UDINT2:UDINT
	VAR_INPUT
		X :	TIME;
	END_VAR

	TIME_TO_UDINT2 := DINT_TO_UDINT(TIME_TO_DINT(X));
END_FUNCTION

FUNCTION_BLOCK MOON_PHASE_Block

	VAR_INPUT
		XDT :	UDINT;
		SCALE :	BYTE := BYTE#12;
		UPDATE :	TIME := T#1h;
	END_VAR

	VAR_OUTPUT
		PHASE :	BYTE;
	END_VAR

	VAR
		x :	UDINT;
		last_dt :	UDINT;
	END_VAR

	IF XDT - last_dt > TIME_TO_UDINT2(UPDATE) THEN
		x := (XDT - UDINT#603240) MOD UDINT#2551392;
		PHASE := UDINT_TO_BYTE(BYTE_TO_UDINT(SCALE) * x / UDINT#2551392) ;
		last_dt := XDT;
	END_IF;

END_FUNCTION_BLOCK

PROGRAM program0
	VAR
		XDT :	UDINT;
		SCALE :	BYTE := BYTE#12;
		UPDATE :	TIME := T#1h;
		PHASE :	BYTE;

		func_block : MOON_PHASE_Block;
	END_VAR
	func_block.XDT := XDT;
	func_block.SCALE := SCALE;
	func_block.UPDATE := UPDATE;

	func_block();
  	PHASE  := func_block.PHASE;
END_PROGRAM

CONFIGURATION Config0
	RESOURCE Res0 ON PLC
		TASK task0(INTERVAL := T#20ms,PRIORITY := 0);
		PROGRAM instance0 WITH task0 : program0;
	END_RESOURCE
END_CONFIGURATION

(* ---- NET_VAR_BOOL8.ST ---- *)
TYPE

	oscat_NW_BUF_LONG  : ARRAY [0..4095] OF BYTE;

	oscat_NETWORK_BUFFER :
	STRUCT
		SIZE   : UINT;
		BUFFER : oscat_NW_BUF_LONG;
	END_STRUCT;

END_TYPE

TYPE oscat_NET_VAR_DATA :
	STRUCT
		CYCLE : UDINT;
		STATE : BYTE;
		INDEX : INT;
		ID_MAX : USINT;
		ERROR_ID : BYTE;
		BUF_SIZE : UINT;
		S_BUF : oscat_NETWORK_BUFFER;
		R_BUF : oscat_NETWORK_BUFFER;
	END_STRUCT;
END_TYPE

FUNCTION BIT_OF_DWORD : BOOL
  VAR_INPUT
    IN : DWORD;
    N : INT;
  END_VAR

  BIT_OF_DWORD := (SHR(in,N) AND 16#00000001) > 0;
END_FUNCTION

FUNCTION_BLOCK BYTE_TO_BITS_Block
	VAR_INPUT
		IN :	BYTE;
	END_VAR

	VAR_OUTPUT
		B0 :	BOOL;
		B1 :	BOOL;
		B2 :	BOOL;
		B3 :	BOOL;
		B4 :	BOOL;
		B5 :	BOOL;
		B6 :	BOOL;
		B7 :	BOOL;
	END_VAR

	B0 := BIT_OF_DWORD(BYTE_TO_DWORD(IN),0); (* IN.X0 *)
	B1 := BIT_OF_DWORD(BYTE_TO_DWORD(IN),1); (* IN.X1 *)
	B2 := BIT_OF_DWORD(BYTE_TO_DWORD(IN),2); (* IN.X2 *)
	B3 := BIT_OF_DWORD(BYTE_TO_DWORD(IN),3); (* IN.X3 *)
	B4 := BIT_OF_DWORD(BYTE_TO_DWORD(IN),4); (* IN.X4 *)
	B5 := BIT_OF_DWORD(BYTE_TO_DWORD(IN),5); (* IN.X5 *)
	B6 := BIT_OF_DWORD(BYTE_TO_DWORD(IN),6); (* IN.X6 *)
	B7 := BIT_OF_DWORD(BYTE_TO_DWORD(IN),7); (* IN.X7 *)
END_FUNCTION_BLOCK

FUNCTION BYTE_OF_BIT:BYTE
	VAR_INPUT
		B0 :	BOOL;
		B1 :	BOOL;
		B2 :	BOOL;
		B3 :	BOOL;
		B4 :	BOOL;
		B5 :	BOOL;
		B6 :	BOOL;
		B7 :	BOOL;
	END_VAR
	Byte_of_bit := SHL(SHL(SHL(SHL(SHL(SHL(SHL(BOOL_TO_BYTE(B7),1) OR BOOL_TO_BYTE(B6),1)
	OR BOOL_TO_BYTE(B5),1) OR BOOL_TO_BYTE(B4),1) OR BOOL_TO_BYTE(B3),1) OR BOOL_TO_BYTE(B2),1)
	OR BOOL_TO_BYTE(B1),1) OR BOOL_TO_BYTE(B0);
END_FUNCTION

FUNCTION_BLOCK NET_VAR_BOOL8_Block

	VAR_INPUT
		IN1 :	BOOL;
		IN2 :	BOOL;
		IN3 :	BOOL;
		IN4 :	BOOL;
		IN5 :	BOOL;
		IN6 :	BOOL;
		IN7 :	BOOL;
		IN8 :	BOOL;
	END_VAR

	VAR_OUTPUT
		OUT1 :	BOOL;
		OUT2 :	BOOL;
		OUT3 :	BOOL;
		OUT4 :	BOOL;
		OUT5 :	BOOL;
		OUT6 :	BOOL;
		OUT7 :	BOOL;
		OUT8 :	BOOL;
		ID :	BYTE;
	END_VAR

	VAR_IN_OUT
		X :	oscat_NET_VAR_DATA;
	END_VAR

	VAR
		init :	BOOL;
		index :	INT;
		index2 :	INT;
		_BYTE_TO_BITS :	BYTE_TO_BITS_Block;
	END_VAR

	IF NOT init THEN
		init := TRUE;
		X.ID_MAX := X.ID_MAX + USINT#1;
		ID := USINT_TO_BYTE(X.ID_MAX);
	END_IF;

	IF X.STATE > BYTE#0 AND X.ERROR_ID = BYTE#0 THEN
		index := X.index;
		IF INT_TO_UINT(index + 3) > X.BUF_SIZE THEN
			X.ERROR_ID := ID;
		ELSE
			IF X.STATE = BYTE#1 THEN
				X.S_BUF.BUFFER[index] := ID;
				index := index + 1;
				X.S_BUF.BUFFER[index] := BYTE#4;
				index := index + 1;
				X.S_BUF.BUFFER[index] := BYTE_OF_BIT(IN1,IN2,IN3,IN4,IN5,IN6,IN7,IN8);
				index := index + 1;

			ELSIF X.STATE = BYTE#2 THEN
				index2 := index + 1;
				IF X.R_BUF.BUFFER[index] <> ID OR X.R_BUF.BUFFER[index2] <> BYTE#4 THEN
					X.ERROR_ID := ID;
				ELSE
					index := index + 2;
					_BYTE_TO_BITS(IN:=X.R_BUF.BUFFER[index]);
					OUT1 := _BYTE_TO_BITS.B0;
					OUT2 := _BYTE_TO_BITS.B1;
					OUT3 := _BYTE_TO_BITS.B2;
					OUT4 := _BYTE_TO_BITS.B3;
					OUT5 := _BYTE_TO_BITS.B4;
					OUT6 := _BYTE_TO_BITS.B5;
					OUT7 := _BYTE_TO_BITS.B6;
					OUT8 := _BYTE_TO_BITS.B7;
					index := index + 1;
				END_IF;
			END_IF;
			X.index := index;
		END_IF;
	END_IF;

END_FUNCTION_BLOCK

PROGRAM program0
	VAR
		IN1 :	BOOL;
		IN2 :	BOOL;
		IN3 :	BOOL;
		IN4 :	BOOL;
		IN5 :	BOOL;
		IN6 :	BOOL;
		IN7 :	BOOL;
		IN8 :	BOOL;
		OUT1 :	BOOL;
		OUT2 :	BOOL;
		OUT3 :	BOOL;
		OUT4 :	BOOL;
		OUT5 :	BOOL;
		OUT6 :	BOOL;
		OUT7 :	BOOL;
		OUT8 :	BOOL;
		ID :	BYTE;
		X :	oscat_NET_VAR_DATA;

		func_block : NET_VAR_BOOL8_Block;
	END_VAR
	func_block.IN1 := IN1;
	func_block.IN2 := IN2;
	func_block.IN3 := IN3;
	func_block.IN4 := IN4;
	func_block.IN5 := IN5;
	func_block.IN6 := IN6;
	func_block.IN7 := IN7;
	func_block.IN8 := IN8;
	func_block.X := X;

	func_block();
  	OUT1  := func_block.OUT1;
	OUT2  := func_block.OUT2;
	OUT3  := func_block.OUT3;
	OUT4  := func_block.OUT4;
	OUT5  := func_block.OUT5;
	OUT6  := func_block.OUT6;
	OUT7  := func_block.OUT7;
	OUT8  := func_block.OUT8;
	ID  := func_block.ID;
	X  := func_block.X;
END_PROGRAM

CONFIGURATION Config0
	RESOURCE Res0 ON PLC
		TASK task0(INTERVAL := T#20ms,PRIORITY := 0);
		PROGRAM instance0 WITH task0 : program0;
	END_RESOURCE
END_CONFIGURATION

(* ---- NET_VAR_BUFFER.ST ---- *)
TYPE
	oscat_aB1_64 : ARRAY[1..64] OF BYTE;
END_TYPE

TYPE

	oscat_NW_BUF_LONG  : ARRAY [0..4095] OF BYTE;

	oscat_NETWORK_BUFFER :
	STRUCT
		SIZE   : UINT;
		BUFFER : oscat_NW_BUF_LONG;
	END_STRUCT;

END_TYPE

TYPE oscat_NET_VAR_DATA :
	STRUCT
		CYCLE : UDINT;
		STATE : BYTE;
		INDEX : INT;
		ID_MAX : USINT;
		ERROR_ID : BYTE;
		BUF_SIZE : UINT;
		S_BUF : oscat_NETWORK_BUFFER;
		R_BUF : oscat_NETWORK_BUFFER;
	END_STRUCT;
END_TYPE

FUNCTION_BLOCK NET_VAR_BUFFER_Block

	VAR_OUTPUT
		ID :	BYTE;
	END_VAR

	VAR_IN_OUT
		BUF_IN :	oscat_aB1_64;
		BUF_OUT :	oscat_aB1_64;
		X :	oscat_NET_VAR_DATA;
	END_VAR

	VAR
		size :	INT;
		init :	BOOL;
		index :	INT;
		index2 :	INT;
	END_VAR

	IF NOT init THEN
		init := TRUE;
		X.ID_MAX := X.ID_MAX + USINT#1;
		ID := USINT_TO_BYTE(X.ID_MAX);
	END_IF;

	IF X.STATE > BYTE#0 AND X.ERROR_ID = BYTE#0 THEN
		index := X.index;
		IF X.STATE = BYTE#1 THEN
			size := 64;
			IF INT_TO_UINT(index + 3 + size) > X.BUF_SIZE THEN
				X.ERROR_ID := ID;
			ELSE
				X.S_BUF.BUFFER[index] := ID;
				index := index + 1;
				X.S_BUF.BUFFER[index] := BYTE#20;
				index := index + 1;
				X.S_BUF.BUFFER[index] := INT_TO_BYTE(size);
				index := index + 1;
				FOR index2 := 1 TO size DO
					X.S_BUF.BUFFER[index] := BUF_IN[index2];
					index := index + 1;
				END_FOR;
			END_IF;
		ELSIF X.STATE = BYTE#2 THEN
			index2 := index + 1;
			IF X.R_BUF.BUFFER[index] <> ID OR X.R_BUF.BUFFER[index2] <> BYTE#20 THEN
				X.ERROR_ID := ID;
			ELSE
				index := index + 2;
				size := BYTE_TO_INT(X.R_BUF.BUFFER[index]);
				index := index + 1;
				FOR index2 := 1 TO size DO
					BUF_OUT[index2] := X.R_BUF.BUFFER[index];
					index := index + 1;
				END_FOR;
			END_IF;
		END_IF;
		X.index := index;
	END_IF;

END_FUNCTION_BLOCK

PROGRAM program0
	VAR
		BUF_IN :	oscat_aB1_64;
		BUF_OUT :	oscat_aB1_64;
		X :	oscat_NET_VAR_DATA;
		ID :	BYTE;

		func_block : NET_VAR_BUFFER_Block;
	END_VAR
	func_block.BUF_IN := BUF_IN;
	func_block.BUF_OUT := BUF_OUT;
	func_block.X := X;

	func_block();
  	BUF_IN  := func_block.BUF_IN;
	BUF_OUT  := func_block.BUF_OUT;
	X  := func_block.X;
	ID  := func_block.ID;

END_PROGRAM

CONFIGURATION Config0
	RESOURCE Res0 ON PLC
		TASK task0(INTERVAL := T#20ms,PRIORITY := 0);
		PROGRAM instance0 WITH task0 : program0;
	END_RESOURCE
END_CONFIGURATION

(* ---- NET_VAR_DWORD8.ST ---- *)
TYPE
	oscat_nv_dw : ARRAY[1..8] OF DWORD;
END_TYPE

TYPE

	oscat_NW_BUF_LONG  : ARRAY [0..4095] OF BYTE;

	oscat_NETWORK_BUFFER :
	STRUCT
		SIZE   : UINT;
		BUFFER : oscat_NW_BUF_LONG;
	END_STRUCT;

END_TYPE

TYPE oscat_NET_VAR_DATA :
	STRUCT
		CYCLE : UDINT;
		STATE : BYTE;
		INDEX : INT;
		ID_MAX : USINT;
		ERROR_ID : BYTE;
		BUF_SIZE : UINT;
		S_BUF : oscat_NETWORK_BUFFER;
		R_BUF : oscat_NETWORK_BUFFER;
	END_STRUCT;
END_TYPE

FUNCTION_BLOCK NET_VAR_DWORD8_Block

	VAR_INPUT
		IN1 :	DWORD;
		IN2 :	DWORD;
		IN3 :	DWORD;
		IN4 :	DWORD;
		IN5 :	DWORD;
		IN6 :	DWORD;
		IN7 :	DWORD;
		IN8 :	DWORD;
	END_VAR

	VAR_OUTPUT
		OUT1 :	DWORD;
		OUT2 :	DWORD;
		OUT3 :	DWORD;
		OUT4 :	DWORD;
		OUT5 :	DWORD;
		OUT6 :	DWORD;
		OUT7 :	DWORD;
		OUT8 :	DWORD;
		ID :	BYTE;
	END_VAR

	VAR_IN_OUT
		X :	oscat_NET_VAR_DATA;
	END_VAR

	VAR
		init :	BOOL;
		i :	INT;
		i2 :	INT;
		index :	INT;
		index2 :	INT;
		ra :	oscat_nv_dw;
	END_VAR

	IF NOT init THEN
		init := TRUE;
		X.ID_MAX := X.ID_MAX + USINT#1;
		ID := USINT_TO_BYTE(X.ID_MAX);
	END_IF;

	IF X.STATE > BYTE#0 AND X.ERROR_ID = BYTE#0 THEN
		index := X.index;
		IF INT_TO_UINT(index + 34) > X.BUF_SIZE THEN
			X.ERROR_ID := ID;
		ELSE
			IF X.STATE = BYTE#1 THEN
				ra[1] := IN1;
				ra[2] := IN2;
				ra[3] := IN3;
				ra[4] := IN4;
				ra[5] := IN5;
				ra[6] := IN6;
				ra[7] := IN7;
				ra[8] := IN8;
				X.S_BUF.BUFFER[index] := ID;
				index := index + 1;
				X.S_BUF.BUFFER[index] := BYTE#13;
				index := index + 1;
				FOR i2 := 1 TO 8 DO
					FOR i := 1 TO 4 DO
						X.S_BUF.BUFFER[index] := DWORD_TO_BYTE(ra[i2]);
						ra[i2] := ROR(ra[i2],8);
						index := index + 1;
					END_FOR;
				END_FOR;

			ELSIF X.STATE = BYTE#2 THEN
				index2 := index + 1;
				IF X.R_BUF.BUFFER[index] <> ID OR X.R_BUF.BUFFER[index2] <> BYTE#13 THEN
					X.ERROR_ID := ID;
				ELSE
					index := index + 2;
					FOR i2 := 1 TO 8 DO
						ra[i2] := DWORD#0;
						FOR i := 1 TO 4 DO
							ra[i2] := ra[i2] OR BYTE_TO_DWORD(X.R_BUF.BUFFER[index]);
							ra[i2] := ROR(ra[i2],8);
							index := index + 1;
						END_FOR;
					END_FOR;
					OUT1 := ra[1];
					OUT2 := ra[2];
					OUT3 := ra[3];
					OUT4 := ra[4];
					OUT5 := ra[5];
					OUT6 := ra[6];
					OUT7 := ra[7];
					OUT8 := ra[8];
				END_IF;
			END_IF;
			X.index := index;
		END_IF;
	END_IF;

END_FUNCTION_BLOCK

PROGRAM program0
	VAR
		IN1 :	DWORD;
		IN2 :	DWORD;
		IN3 :	DWORD;
		IN4 :	DWORD;
		IN5 :	DWORD;
		IN6 :	DWORD;
		IN7 :	DWORD;
		IN8 :	DWORD;
		OUT1 :	DWORD;
		OUT2 :	DWORD;
		OUT3 :	DWORD;
		OUT4 :	DWORD;
		OUT5 :	DWORD;
		OUT6 :	DWORD;
		OUT7 :	DWORD;
		OUT8 :	DWORD;
		ID :	BYTE;
		X :	oscat_NET_VAR_DATA;

		func_block : NET_VAR_DWORD8_Block;
	END_VAR
	func_block.IN1 := IN1;
	func_block.IN2 := IN2;
	func_block.IN3 := IN3;
	func_block.IN4 := IN4;
	func_block.IN5 := IN5;
	func_block.IN6 := IN6;
	func_block.IN7 := IN7;
	func_block.IN8 := IN8;
	func_block.X := X;

	func_block();
  	OUT1  := func_block.OUT1;
	OUT2  := func_block.OUT2;
	OUT3  := func_block.OUT3;
	OUT4  := func_block.OUT4;
	OUT5  := func_block.OUT5;
	OUT6  := func_block.OUT6;
	OUT7  := func_block.OUT7;
	OUT8  := func_block.OUT8;
	ID  := func_block.ID;
	X  := func_block.X;
END_PROGRAM

CONFIGURATION Config0
	RESOURCE Res0 ON PLC
		TASK task0(INTERVAL := T#20ms,PRIORITY := 0);
		PROGRAM instance0 WITH task0 : program0;
	END_RESOURCE
END_CONFIGURATION

(* ---- ONTIME.ST ---- *)
FUNCTION_BLOCK T_PLC_MS_block
	VAR_OUTPUT
		T_PLC_MS :	UDINT;
	END_VAR

	VAR_EXTERNAL
		PLC_TICKS_PER_SEC :	INT;
		PLC_SYS_TICK_CNT :	DINT;
	END_VAR

	VAR
		debug :	BOOL;(*Debug-Mode ON / OFF*)
		N :	INT;(*Debug-Faktor*)
		Offset :	UDINT;(*Debug-Offset*)
		temp :	DWORD := DWORD#1;(*Debug-Offset*)
		mode :	BOOL;(*modus*)
		faktor :	UDINT;(*Systemtakt-Faktor*)
		init :	BOOL;
		v_plc_ticks_per_sec :	UDINT;
		base :	UDINT := UDINT#1000;
	END_VAR

	IF init = FALSE THEN
		v_plc_ticks_per_sec := INT_TO_UDINT(PLC_TICKS_PER_SEC);
		IF v_plc_ticks_per_sec = UDINT#1024 THEN
			faktor := UDINT#1;
			mode := FALSE;
		ELSIF v_plc_ticks_per_sec > UDINT#0 THEN
			IF v_plc_ticks_per_sec <= base THEN
				faktor := base / v_plc_ticks_per_sec;
				mode := FALSE;
			ELSE
				faktor := v_plc_ticks_per_sec / base;
				mode := TRUE;
			END_IF;
		ELSE
			faktor := UDINT#1;
		END_IF;
		init := TRUE;
	END_IF;

	IF mode THEN
		T_PLC_MS := DINT_TO_UDINT(PLC_SYS_TICK_CNT) / faktor;
	ELSE
		T_PLC_MS := DINT_TO_UDINT(PLC_SYS_TICK_CNT) * faktor;
	END_IF;

	IF debug THEN
		T_PLC_MS := (DWORD_TO_UDINT(SHL(UDINT_TO_DWORD(T_PLC_MS),N) OR SHL(temp,N)) - UDINT#1) + Offset;
	END_IF;

END_FUNCTION_BLOCK

FUNCTION_BLOCK ONTIME_Block

	VAR_INPUT
		IN :	BOOL;
		RST :	BOOL;
	END_VAR

	VAR_IN_OUT
		SECONDS :	UDINT;
		CYCLES :	UDINT;
	END_VAR

	VAR
		tx :	UDINT;
		last :	UDINT;
		edge :	BOOL;
		init :	BOOL;
		ms :	UDINT;
		T_PLC_MS :	T_PLC_MS_Block;
	END_VAR

	T_PLC_MS();
	tx:= T_PLC_MS.T_PLC_MS;

	IF NOT init THEN
		init := TRUE;
		last := tx;
		ms := UDINT#0;
	END_IF;
	IF RST THEN
		SECONDS := UDINT#0;
		CYCLES := UDINT#0;
		last := tx;
		ms := UDINT#0;
	ELSIF IN THEN
		(* add the current milliseconds *)
		ms := (tx - last) + ms;
		IF ms >= UDINT#1000 THEN
			seconds := seconds + UDINT#1;
			ms := ms - UDINT#1000;
		END_IF;
		cycles := cycles + BOOL_TO_UDINT(NOT edge);
	END_IF;
	last := tx;
	edge := in;

END_FUNCTION_BLOCK

PROGRAM program0
	VAR
		IN :	BOOL;
		RST :	BOOL;
		SECONDS :	UDINT;
		CYCLES :	UDINT;
		func_block : ONTIME_Block;
	END_VAR
	func_block.IN := IN;
	func_block.RST := RST;
	func_block();
	SECONDS  := func_block.SECONDS;
	CYCLES  := func_block.CYCLES;
END_PROGRAM

CONFIGURATION Config0
	VAR_GLOBAL
		PLC_TICKS_PER_SEC :	INT;
		PLC_SYS_TICK_CNT :	DINT;
	END_VAR
  	RESOURCE Res0 ON PLC
    	TASK task0(INTERVAL := T#20ms,PRIORITY := 0);
    	PROGRAM instance0 WITH task0 : program0;
  	END_RESOURCE
END_CONFIGURATION

(* ---- PARSET.ST ---- *)
TYPE
	oscat_parset_X              : ARRAY [1..4]    OF REAL;
	oscat_parset                : ARRAY [0..3]    OF oscat_parset_X := [0,0,0,0];
END_TYPE

FUNCTION TIME_TO_UDINT2:UDINT
	VAR_INPUT
		X :	TIME;
	END_VAR

	TIME_TO_UDINT2 := DINT_TO_UDINT(TIME_TO_DINT(X));
END_FUNCTION

FUNCTION _BYTE_TO_INT:INT
	VAR_INPUT
		IN :	BYTE;
	END_VAR

	_BYTE_TO_INT := USINT_TO_INT(BYTE_TO_USINT(IN));
END_FUNCTION

FUNCTION BIT_OF_DWORD : BOOL
  VAR_INPUT
    IN : DWORD;
    N : INT;
  END_VAR

  BIT_OF_DWORD := (SHR(in,N) AND 16#00000001) > 0;
  (* from OSCAT library; www.oscat.de  *)
END_FUNCTION

FUNCTION BIT_LOAD_B:BYTE
	VAR_INPUT
		IN :	BYTE;
		VAL :	BOOL;
		POS :	INT;
	END_VAR

	IF VAL THEN
		BIT_LOAD_B := in OR SHL(BYTE#1,pos);
	ELSE
		BIT_LOAD_B := in AND (NOT SHL(BYTE#1,pos));
	END_IF;
END_FUNCTION

FUNCTION_BLOCK T_PLC_MS_block
	VAR_OUTPUT
		T_PLC_MS :	UDINT;
	END_VAR

	VAR_EXTERNAL
		PLC_TICKS_PER_SEC :	INT;
		PLC_SYS_TICK_CNT :	DINT;
	END_VAR

	VAR
		debug :	BOOL;(*Debug-Mode ON / OFF*)
		N :	INT;(*Debug-Faktor*)
		Offset :	UDINT;(*Debug-Offset*)
		temp :	DWORD := DWORD#1;(*Debug-Offset*)
		mode :	BOOL;(*modus*)
		faktor :	UDINT;(*Systemtakt-Faktor*)
		init :	BOOL;
		v_plc_ticks_per_sec :	UDINT;
		base :	UDINT := UDINT#1000;
	END_VAR

	IF init = FALSE THEN
		v_plc_ticks_per_sec := INT_TO_UDINT(PLC_TICKS_PER_SEC);
		IF v_plc_ticks_per_sec = UDINT#1024 THEN
			faktor := UDINT#1;
			mode := FALSE;
		ELSIF v_plc_ticks_per_sec > UDINT#0 THEN
			IF v_plc_ticks_per_sec <= base THEN
				faktor := base / v_plc_ticks_per_sec;
				mode := FALSE;
			ELSE
				faktor := v_plc_ticks_per_sec / base;
				mode := TRUE;
			END_IF;
		ELSE
			faktor := UDINT#1;
		END_IF;
		init := TRUE;
	END_IF;

	IF mode THEN
		T_PLC_MS := DINT_TO_UDINT(PLC_SYS_TICK_CNT) / faktor;
	ELSE
		T_PLC_MS := DINT_TO_UDINT(PLC_SYS_TICK_CNT) * faktor;
	END_IF;

	IF debug THEN
		T_PLC_MS := (DWORD_TO_UDINT(SHL(UDINT_TO_DWORD(T_PLC_MS),N) OR SHL(temp,N)) - UDINT#1) + Offset;
	END_IF;
END_FUNCTION_BLOCK

FUNCTION_BLOCK PARSET_Block

	VAR_INPUT
		A0 :	BOOL;
		A1 :	BOOL;
		X01 :	REAL;
		X02 :	REAL;
		X03 :	REAL;
		X04 :	REAL;
		X11 :	REAL;
		X12 :	REAL;
		X13 :	REAL;
		X14 :	REAL;
		X21 :	REAL;
		X22 :	REAL;
		X23 :	REAL;
		X24 :	REAL;
		X31 :	REAL;
		X32 :	REAL;
		X33 :	REAL;
		X34 :	REAL;
		TC :	TIME;
	END_VAR

	VAR_OUTPUT
		P1 :	REAL;
		P2 :	REAL;
		P3 :	REAL;
		P4 :	REAL;
	END_VAR

	VAR
		X :	oscat_parset;
		S1 :	REAL;
		S2 :	REAL;
		S3 :	REAL;
		S4 :	REAL;
		tx :	UDINT;
		last :	UDINT;
		start :	BOOL;
		set :	BYTE;
		set2 :	INT;
		init :	BOOL;
		T_PLC_MS :	T_PLC_MS_Block;
	END_VAR

	(*@KEY@: WORKSHEET
	NAME: PARSET
	IEC_LANGUAGE: ST
	*)
	(* read system_time *)
	T_PLC_MS();
	tx:= T_PLC_MS.T_PLC_MS;

	(* init sequence *)
	IF NOT init THEN
		set:=BIT_LOAD_B(set,NOT A0,0); (* set.X0 := NOT A0; *)
		init := TRUE;
		X[0][1] := X01;
		X[0][2] := X02;
		X[0][3] := X03;
		X[0][4] := X04;
		X[1][1] := X11;
		X[1][2] := X12;
		X[1][3] := X13;
		X[1][4] := X14;
		X[2][1] := X21;
		X[2][2] := X22;
		X[2][3] := X23;
		X[2][4] := X24;
		X[3][1] := X31;
		X[3][2] := X32;
		X[3][3] := X33;
		X[3][4] := X34;
		P1 := X01;
		P2 := X02;
		P3 := X03;
		P4 := X04;
	END_IF;

	(* check for input change *)
	IF (A0 XOR BIT_OF_DWORD(BYTE_TO_DWORD(set),0)) OR (A1 XOR BIT_OF_DWORD(BYTE_TO_DWORD(set),1)) THEN  (* set.X0  ,  set.X1 *)
		(* a new set is selected *)
		set := BIT_LOAD_B(set,A0,0); (* set.X0 := A0; *)
		set := BIT_LOAD_B(set,A1,1); (* set.X1 := A1; *)

		IF tc > t#0s THEN
			start := TRUE;
			last := tx;
			(* save the step speed for the output changes in S *)
			set2 := _BYTE_TO_INT(set);
			S1 := (X[set2][1] - P1)/TIME_TO_REAL(tc);
			S2 := (X[set2][2] - P2)/TIME_TO_REAL(tc);
			S3 := (X[set2][3] - P3)/TIME_TO_REAL(tc);
			S4 := (X[set2][4] - P4)/TIME_TO_REAL(tc);
		END_IF;
	ELSIF start AND tx - last < TIME_TO_UDINT2(tc) THEN
		(* ramp the outputs to the new value *)
		set2 := _BYTE_TO_INT(set);
		P1 := X[set2][1] - S1*(TIME_TO_REAL(Tc) - UDINT_TO_REAL(tx + last));
		P2 := X[set2][2] - S2*(TIME_TO_REAL(Tc) - UDINT_TO_REAL(tx + last));
		P3 := X[set2][3] - S3*(TIME_TO_REAL(Tc) - UDINT_TO_REAL(tx + last));
		P4 := X[set2][4] - S4*(TIME_TO_REAL(Tc) - UDINT_TO_REAL(tx + last));
	ELSE
		(* make sure outputs match the correct set values *)
		set2 := _BYTE_TO_INT(set);
		start := FALSE;
		P1 := X[set2][1];
		P2 := X[set2][2];
		P3 := X[set2][3];
		P4 := X[set2][4];
	END_IF;

END_FUNCTION_BLOCK

PROGRAM program0

	VAR
		A0 :	BOOL;
		A1 :	BOOL;
		X01 :	REAL;
		X02 :	REAL;
		X03 :	REAL;
		X04 :	REAL;
		X11 :	REAL;
		X12 :	REAL;
		X13 :	REAL;
		X14 :	REAL;
		X21 :	REAL;
		X22 :	REAL;
		X23 :	REAL;
		X24 :	REAL;
		X31 :	REAL;
		X32 :	REAL;
		X33 :	REAL;
		X34 :	REAL;
		TC :	TIME;

		P1 :	REAL;
		P2 :	REAL;
		P3 :	REAL;
		P4 :	REAL;
		func_block : PARSET_Block;
  	END_VAR
	func_block.A0 := A0;
	func_block.A1 := A1;
	func_block.X01 := X01;
	func_block.X02 := X02;
	func_block.X03 := X03;
	func_block.X04 := X04;
	func_block.X11 := X11;
	func_block.X12 := X12;
	func_block.X13 := X13;
	func_block.X14 := X14;
	func_block.X21 := X21;
	func_block.X22 := X22;
	func_block.X23 := X23;
	func_block.X24 := X24;
	func_block.X31 := X31;
	func_block.X32 := X32;
	func_block.X33 := X33;
	func_block.X34 := X34;
	func_block.TC := TC;
	func_block();
	P1 := func_block.P1;
	P2 := func_block.P2;
	P3 := func_block.P3;
	P4 := func_block.P4;

END_PROGRAM

CONFIGURATION Config0

	VAR_GLOBAL
		PLC_TICKS_PER_SEC :	INT;
		PLC_SYS_TICK_CNT :	DINT;
	END_VAR

  	RESOURCE Res0 ON PLC
    	TASK task0(INTERVAL := T#20ms,PRIORITY := 0);
    	PROGRAM instance0 WITH task0 : program0;
  	END_RESOURCE

END_CONFIGURATION

(* ---- PARSET2.ST ---- *)
TYPE
	oscat_parset_X              : ARRAY [1..4]    OF REAL;
	oscat_parset                : ARRAY [0..3]    OF oscat_parset_X := [0,0,0,0];
END_TYPE

FUNCTION TIME_TO_UDINT2:UDINT
	VAR_INPUT
		X :	TIME;
	END_VAR

	TIME_TO_UDINT2 := DINT_TO_UDINT(TIME_TO_DINT(X));
END_FUNCTION

FUNCTION _BYTE_TO_INT:INT
	VAR_INPUT
		IN :	BYTE;
	END_VAR

	_BYTE_TO_INT := USINT_TO_INT(BYTE_TO_USINT(IN));
END_FUNCTION

FUNCTION BIT_OF_DWORD : BOOL
  VAR_INPUT
    IN : DWORD;
    N : INT;
  END_VAR

  BIT_OF_DWORD := (SHR(in,N) AND 16#00000001) > 0;
  (* from OSCAT library; www.oscat.de  *)
END_FUNCTION

FUNCTION BIT_LOAD_B:BYTE
	VAR_INPUT
		IN :	BYTE;
		VAL :	BOOL;
		POS :	INT;
	END_VAR

	IF VAL THEN
		BIT_LOAD_B := in OR SHL(BYTE#1,pos);
	ELSE
		BIT_LOAD_B := in AND (NOT SHL(BYTE#1,pos));
	END_IF;
END_FUNCTION

FUNCTION_BLOCK T_PLC_MS_block
	VAR_OUTPUT
		T_PLC_MS :	UDINT;
	END_VAR

	VAR_EXTERNAL
		PLC_TICKS_PER_SEC :	INT;
		PLC_SYS_TICK_CNT :	DINT;
	END_VAR

	VAR
		debug :	BOOL;(*Debug-Mode ON / OFF*)
		N :	INT;(*Debug-Faktor*)
		Offset :	UDINT;(*Debug-Offset*)
		temp :	DWORD := DWORD#1;(*Debug-Offset*)
		mode :	BOOL;(*modus*)
		faktor :	UDINT;(*Systemtakt-Faktor*)
		init :	BOOL;
		v_plc_ticks_per_sec :	UDINT;
		base :	UDINT := UDINT#1000;
	END_VAR

	IF init = FALSE THEN
		v_plc_ticks_per_sec := INT_TO_UDINT(PLC_TICKS_PER_SEC);
		IF v_plc_ticks_per_sec = UDINT#1024 THEN
			faktor := UDINT#1;
			mode := FALSE;
		ELSIF v_plc_ticks_per_sec > UDINT#0 THEN
			IF v_plc_ticks_per_sec <= base THEN
				faktor := base / v_plc_ticks_per_sec;
				mode := FALSE;
			ELSE
				faktor := v_plc_ticks_per_sec / base;
				mode := TRUE;
			END_IF;
		ELSE
			faktor := UDINT#1;
		END_IF;
		init := TRUE;
	END_IF;

	IF mode THEN
		T_PLC_MS := DINT_TO_UDINT(PLC_SYS_TICK_CNT) / faktor;
	ELSE
		T_PLC_MS := DINT_TO_UDINT(PLC_SYS_TICK_CNT) * faktor;
	END_IF;

	IF debug THEN
		T_PLC_MS := (DWORD_TO_UDINT(SHL(UDINT_TO_DWORD(T_PLC_MS),N) OR SHL(temp,N)) - UDINT#1) + Offset;
	END_IF;
END_FUNCTION_BLOCK

FUNCTION_BLOCK PARSET_Block

	VAR_INPUT
		A0 :	BOOL;
		A1 :	BOOL;
		X01 :	REAL;
		X02 :	REAL;
		X03 :	REAL;
		X04 :	REAL;
		X11 :	REAL;
		X12 :	REAL;
		X13 :	REAL;
		X14 :	REAL;
		X21 :	REAL;
		X22 :	REAL;
		X23 :	REAL;
		X24 :	REAL;
		X31 :	REAL;
		X32 :	REAL;
		X33 :	REAL;
		X34 :	REAL;
		TC :	TIME;
	END_VAR

	VAR_OUTPUT
		P1 :	REAL;
		P2 :	REAL;
		P3 :	REAL;
		P4 :	REAL;
	END_VAR

	VAR
		X :	oscat_parset;
		S1 :	REAL;
		S2 :	REAL;
		S3 :	REAL;
		S4 :	REAL;
		tx :	UDINT;
		last :	UDINT;
		start :	BOOL;
		set :	BYTE;
		set2 :	INT;
		init :	BOOL;
		T_PLC_MS :	T_PLC_MS_Block;
	END_VAR

	(*@KEY@: WORKSHEET
	NAME: PARSET
	IEC_LANGUAGE: ST
	*)
	(* read system_time *)
	T_PLC_MS();
	tx:= T_PLC_MS.T_PLC_MS;

	(* init sequence *)
	IF NOT init THEN
		set:=BIT_LOAD_B(set,NOT A0,0); (* set.X0 := NOT A0; *)
		init := TRUE;
		X[0][1] := X01;
		X[0][2] := X02;
		X[0][3] := X03;
		X[0][4] := X04;
		X[1][1] := X11;
		X[1][2] := X12;
		X[1][3] := X13;
		X[1][4] := X14;
		X[2][1] := X21;
		X[2][2] := X22;
		X[2][3] := X23;
		X[2][4] := X24;
		X[3][1] := X31;
		X[3][2] := X32;
		X[3][3] := X33;
		X[3][4] := X34;
		P1 := X01;
		P2 := X02;
		P3 := X03;
		P4 := X04;
	END_IF;

	(* check for input change *)
	IF (A0 XOR BIT_OF_DWORD(BYTE_TO_DWORD(set),0)) OR (A1 XOR BIT_OF_DWORD(BYTE_TO_DWORD(set),1)) THEN  (* set.X0  ,  set.X1 *)
		(* a new set is selected *)
		set := BIT_LOAD_B(set,A0,0); (* set.X0 := A0; *)
		set := BIT_LOAD_B(set,A1,1); (* set.X1 := A1; *)

		IF tc > t#0s THEN
			start := TRUE;
			last := tx;
			(* save the step speed for the output changes in S *)
			set2 := _BYTE_TO_INT(set);
			S1 := (X[set2][1] - P1)/TIME_TO_REAL(tc);
			S2 := (X[set2][2] - P2)/TIME_TO_REAL(tc);
			S3 := (X[set2][3] - P3)/TIME_TO_REAL(tc);
			S4 := (X[set2][4] - P4)/TIME_TO_REAL(tc);
		END_IF;
	ELSIF start AND tx - last < TIME_TO_UDINT2(tc) THEN
		(* ramp the outputs to the new value *)
		set2 := _BYTE_TO_INT(set);
		P1 := X[set2][1] - S1*(TIME_TO_REAL(Tc) - UDINT_TO_REAL(tx + last));
		P2 := X[set2][2] - S2*(TIME_TO_REAL(Tc) - UDINT_TO_REAL(tx + last));
		P3 := X[set2][3] - S3*(TIME_TO_REAL(Tc) - UDINT_TO_REAL(tx + last));
		P4 := X[set2][4] - S4*(TIME_TO_REAL(Tc) - UDINT_TO_REAL(tx + last));
	ELSE
		(* make sure outputs match the correct set values *)
		set2 := _BYTE_TO_INT(set);
		start := FALSE;
		P1 := X[set2][1];
		P2 := X[set2][2];
		P3 := X[set2][3];
		P4 := X[set2][4];
	END_IF;

END_FUNCTION_BLOCK

FUNCTION_BLOCK PARSET2_Block

	VAR_INPUT
		X :	REAL;
		X01 :	REAL;
		X02 :	REAL;
		X03 :	REAL;
		X04 :	REAL;
		X11 :	REAL;
		X12 :	REAL;
		X13 :	REAL;
		X14 :	REAL;
		X21 :	REAL;
		X22 :	REAL;
		X23 :	REAL;
		X24 :	REAL;
		X31 :	REAL;
		X32 :	REAL;
		X33 :	REAL;
		X34 :	REAL;
		L1 :	REAL;
		L2 :	REAL;
		L3 :	REAL;
		TC :	TIME;
	END_VAR

	VAR_OUTPUT
		P1 :	REAL;
		P2 :	REAL;
		P3 :	REAL;
		P4 :	REAL;
	END_VAR

	VAR
		Pset :	PARSET_Block;
		init :	BOOL;
	END_VAR

	IF NOT init THEN
		init := TRUE;
		pset(TC:=TC, X01:=X01, X02:=X02, X03:=X03, X04:=X04, X11:=X11, X12:=X12, X13:=X13, X14:=X14, X21:=X21, X22:=X22, X23:=X23, X24:=X24, X31:=X31, X32:=X32, X33:=X33, X34:=X34);
	END_IF;
	IF ABS(X) < L1 THEN
		pset(A0 := FALSE, A1 := FALSE);
	ELSIF ABS(X) < L2 THEN
		pset(A0 := TRUE, A1 := FALSE);
	ELSIF ABS(x) < L3 THEN
		pset(A0 := FALSE, A1 := TRUE);
	ELSE
		pset(A0 := TRUE, A1 := TRUE);
	END_IF;
	P1 := pset.P1;
	P2 := pset.P2;
	P3 := pset.P3;
	P4 := pset.P4;

END_FUNCTION_BLOCK

PROGRAM program0

	VAR
		X :	REAL;
		X01 :	REAL;
		X02 :	REAL;
		X03 :	REAL;
		X04 :	REAL;
		X11 :	REAL;
		X12 :	REAL;
		X13 :	REAL;
		X14 :	REAL;
		X21 :	REAL;
		X22 :	REAL;
		X23 :	REAL;
		X24 :	REAL;
		X31 :	REAL;
		X32 :	REAL;
		X33 :	REAL;
		X34 :	REAL;
		L1 :	REAL;
		L2 :	REAL;
		L3 :	REAL;
		TC :	TIME;

		P1 :	REAL;
		P2 :	REAL;
		P3 :	REAL;
		P4 :	REAL;
		func_block : PARSET2_Block;
  	END_VAR
	func_block.X01 := X01;
	func_block.X02 := X02;
	func_block.X03 := X03;
	func_block.X04 := X04;
	func_block.X11 := X11;
	func_block.X12 := X12;
	func_block.X13 := X13;
	func_block.X14 := X14;
	func_block.X21 := X21;
	func_block.X22 := X22;
	func_block.X23 := X23;
	func_block.X24 := X24;
	func_block.X31 := X31;
	func_block.X32 := X32;
	func_block.X33 := X33;
	func_block.X34 := X34;
	func_block.L1 := L1;
	func_block.L2 := L2;
	func_block.L3 := L3;
	func_block.TC := TC;
	func_block();
	P1 := func_block.P1;
	P2 := func_block.P2;
	P3 := func_block.P3;
	P4 := func_block.P4;

END_PROGRAM

CONFIGURATION Config0

	VAR_GLOBAL
		PLC_TICKS_PER_SEC :	INT;
		PLC_SYS_TICK_CNT :	DINT;
	END_VAR

  	RESOURCE Res0 ON PLC
    	TASK task0(INTERVAL := T#20ms,PRIORITY := 0);
    	PROGRAM instance0 WITH task0 : program0;
  	END_RESOURCE

END_CONFIGURATION

(* ---- PERIOD2.ST ---- *)
TYPE
	oscat_PERIOD2_Y             : ARRAY [0..1]    OF UDINT;
	oscat_PERIOD2_X             : ARRAY [0..3]    OF oscat_PERIOD2_Y := [0, 0, 0, 0];
END_TYPE

FUNCTION_BLOCK PERIOD2_Block

	VAR_INPUT
		DP :	oscat_PERIOD2_X;
		DX :	UDINT;
	END_VAR

	VAR_OUTPUT
		PERIOD2 :	BOOL;
	END_VAR

	(*@KEY@: WORKSHEET
	NAME: PERIOD2
	IEC_LANGUAGE: ST
	*)
	PERIOD2 := 	(DX >= DP[0][0] AND DX <= DP[0][1]) OR
				(DX >= DP[1][0] AND DX <= DP[1][1]) OR
				(DX >= DP[2][0] AND DX <= DP[2][1]) OR
				(DX >= DP[3][0] AND DX <= DP[3][1]);

END_FUNCTION_BLOCK

PROGRAM program0

	VAR
		DP :	oscat_PERIOD2_X;
		DX :	UDINT;

		PERIOD2 :	BOOL;
		func_block : PERIOD2_Block;
  	END_VAR

	func_block.DP := DP;
	func_block.DX := DX;
	func_block();
	PERIOD2 := func_block.PERIOD2;

END_PROGRAM

CONFIGURATION Config0

  	RESOURCE Res0 ON PLC
    	TASK task0(INTERVAL := T#20ms,PRIORITY := 0);
    	PROGRAM instance0 WITH task0 : program0;
  	END_RESOURCE

END_CONFIGURATION

(* ---- POLYNOM_INT.ST ---- *)
TYPE
	oscat_Polynom_ARRAY_X       : ARRAY [0..1]    OF REAL;
END_TYPE

TYPE
	oscat_Polynom_XY            : ARRAY [1..5]  OF oscat_Polynom_ARRAY_X := [0, 0, 0, 0, 0];
END_TYPE

FUNCTION_BLOCK POLYNOM_INT_Block

	VAR_INPUT
		X :	REAL;
		XY :	oscat_Polynom_XY;
	END_VAR

	VAR_INPUT
		PTS :	INT;
	END_VAR

	VAR_OUTPUT
		POLYNOM_INT :	REAL;
	END_VAR

	VAR
		XY2 :	oscat_Polynom_XY;
	END_VAR

	VAR
		I :	INT;
		J :	INT;
		J_1 :	INT;
		J_I :	INT;
		INIT :	BOOL;
	END_VAR

	pts := MIN_INT(pts, 5);

	IF (init = FALSE) THEN
		init := TRUE;

		FOR i := 1 TO pts DO
			FOR j := 0 TO 1 DO
					XY2[i][j] := XY[i][j];
			END_FOR;
		END_FOR;

		FOR i := 1 TO pts DO
			J := pts;
			WHILE (J >= i+1) DO
			j_i := j-i;
			j_1 := J-1;
			XY2[j][1] := (XY2[j][1] - XY2[j_1][1]) / (XY2[j][0] - XY2[j_i][0]);
			j := j - 1;
			END_WHILE;
		END_FOR;
	END_IF;

END_FUNCTION_BLOCK

PROGRAM program0

	VAR
		X :	REAL;
		XY :	oscat_Polynom_XY;
		PTS :	INT;

		OUT :	REAL;
		func_block : POLYNOM_INT_Block;
  	END_VAR

	func_block.X := X;
	func_block.XY := XY;
	func_block.PTS := PTS;
	func_block();
	OUT := func_block.POLYNOM_INT;

END_PROGRAM

CONFIGURATION Config0

  	RESOURCE Res0 ON PLC
    	TASK task0(INTERVAL := T#20ms,PRIORITY := 0);
    	PROGRAM instance0 WITH task0 : program0;
  	END_RESOURCE

END_CONFIGURATION

(* ---- PRESSURE.ST ---- *)
FUNCTION_BLOCK PRESSURE_Block

	VAR_INPUT
		MWS :	REAL;
		TORR :	REAL;
		ATT :	REAL;
		ATM :	REAL;
		PA :	REAL;
		BAR :	REAL;
	END_VAR

	VAR_OUTPUT
		YMWS :	REAL;
		YTORR :	REAL;
		YATT :	REAL;
		YATM :	REAL;
		YPA :	REAL;
		YBAR :	REAL;
	END_VAR

	Ybar := bar +
			pa * 1.0E-5 +
			0.980665 * att +
			1.01325 * atm +
			0.001333224 * torr +
			0.0980665 * mws;
	Ymws := ybar * 10.1971621297793;
	Ytorr := ybar * 750.0615050434140;
	Yatt := ybar * 1.0197162129779;
	yatm := ybar * 0.9869232667160;
	Ypa := ybar * 100000.0;

END_FUNCTION_BLOCK

PROGRAM program0

	VAR
		MWS :	REAL;
		TORR :	REAL;
		ATT :	REAL;
		ATM :	REAL;
		PA :	REAL;
		BAR :	REAL;

		YMWS :	REAL;
		YTORR :	REAL;
		YATT :	REAL;
		YATM :	REAL;
		YPA :	REAL;
		YBAR :	REAL;
		func_block : PRESSURE_Block;
  	END_VAR
	func_block.MWS := MWS;
	func_block.TORR := TORR;
	func_block.ATT := ATT;
	func_block.ATM := ATM;
	func_block.PA := PA;
	func_block.BAR := BAR;
	func_block();
	YMWS := func_block.YMWS;
	YTORR := func_block.YTORR;
	YATT := func_block.YATT;
	YATM := func_block.YATM;
	YPA := func_block.YPA;
	YBAR := func_block.YBAR;

END_PROGRAM

CONFIGURATION Config0

  	RESOURCE Res0 ON PLC
    	TASK task0(INTERVAL := T#20ms,PRIORITY := 0);
    	PROGRAM instance0 WITH task0 : program0;
  	END_RESOURCE

END_CONFIGURATION

(* ---- PULSE_LENGTH.ST ---- *)
FUNCTION UDINT_TO_TIME2:TIME

	VAR_INPUT
		IN :	UDINT;
	END_VAR

	UDINT_TO_TIME2 := DINT_TO_TIME(UDINT_TO_DINT(IN));

END_FUNCTION

FUNCTION_BLOCK T_PLC_MS_block
	VAR_OUTPUT
		T_PLC_MS :	UDINT;
	END_VAR

	VAR_EXTERNAL
		PLC_TICKS_PER_SEC :	INT;
		PLC_SYS_TICK_CNT :	DINT;
	END_VAR

	VAR
		debug :	BOOL;(*Debug-Mode ON / OFF*)
		N :	INT;(*Debug-Faktor*)
		Offset :	UDINT;(*Debug-Offset*)
		temp :	DWORD := DWORD#1;(*Debug-Offset*)
		mode :	BOOL;(*modus*)
		faktor :	UDINT;(*Systemtakt-Faktor*)
		init :	BOOL;
		v_plc_ticks_per_sec :	UDINT;
		base :	UDINT := UDINT#1000;
	END_VAR

	IF init = FALSE THEN
		v_plc_ticks_per_sec := INT_TO_UDINT(PLC_TICKS_PER_SEC);
		IF v_plc_ticks_per_sec = UDINT#1024 THEN
			faktor := UDINT#1;
			mode := FALSE;
		ELSIF v_plc_ticks_per_sec > UDINT#0 THEN
			IF v_plc_ticks_per_sec <= base THEN
				faktor := base / v_plc_ticks_per_sec;
				mode := FALSE;
			ELSE
				faktor := v_plc_ticks_per_sec / base;
				mode := TRUE;
			END_IF;
		ELSE
			faktor := UDINT#1;
		END_IF;
		init := TRUE;
	END_IF;

	IF mode THEN
		T_PLC_MS := DINT_TO_UDINT(PLC_SYS_TICK_CNT) / faktor;
	ELSE
		T_PLC_MS := DINT_TO_UDINT(PLC_SYS_TICK_CNT) * faktor;
	END_IF;

	IF debug THEN
		T_PLC_MS := (DWORD_TO_UDINT(SHL(UDINT_TO_DWORD(T_PLC_MS),N) OR SHL(temp,N)) - UDINT#1) + Offset;
	END_IF;

END_FUNCTION_BLOCK

FUNCTION_BLOCK PULSE_LENGTH_Block

	VAR_INPUT
		IN :	BOOL;
		T_SHORT :	TIME := T#100ms;
		T_LONG :	TIME := T#1s;
	END_VAR

	VAR_OUTPUT
		SHORT :	BOOL;
		MIDDLE :	BOOL;
		LONG :	BOOL;
	END_VAR

	VAR
		tx :	TIME;
		tn :	TIME;
		edge :	BOOL;
		T_PLC_MS :	T_PLC_MS_Block;
	END_VAR

	T_PLC_MS();
	tx:= UDINT_TO_TIME(T_PLC_MS.T_PLC_MS);

	short := FALSE;
	Middle := FALSE;
	long := FALSE;

	IF in AND NOT edge THEN
		edge := TRUE;
		tn := tx;

	ELSIF NOT in AND edge THEN
		edge := FALSE;
		tn := tx - tn;
		IF tn < t_short THEN
			short := TRUE;
		ELSIF tn > t_long THEN
			long := TRUE;
		ELSE
			Middle := TRUE;
		END_IF;

	ELSIF in AND tx - tn > t_long THEN
		long := TRUE;
	END_IF;

END_FUNCTION_BLOCK

PROGRAM program0
	VAR
		IN :	BOOL;
		T_SHORT :	TIME := T#100ms;
		T_LONG :	TIME := T#1s;
		SHORT :	BOOL;
		MIDDLE :	BOOL;
		LONG :	BOOL;

		func_block : PULSE_LENGTH_Block;
	END_VAR
	func_block.IN := IN;
	func_block.T_SHORT := T_SHORT;
	func_block.T_LONG := T_LONG ;

	func_block();
	SHORT  := func_block.SHORT;
	MIDDLE  := func_block.MIDDLE;
	LONG  := func_block.LONG;
END_PROGRAM

CONFIGURATION Config0
	VAR_GLOBAL
		PLC_TICKS_PER_SEC :	INT;
		PLC_SYS_TICK_CNT :	DINT;
	END_VAR
  	RESOURCE Res0 ON PLC
    	TASK task0(INTERVAL := T#20ms,PRIORITY := 0);
    	PROGRAM instance0 WITH task0 : program0;
  	END_RESOURCE
END_CONFIGURATION

(* ---- PULSE_T.ST ---- *)
FUNCTION UDINT_TO_TIME2:TIME

	VAR_INPUT
		IN :	UDINT;
	END_VAR

	UDINT_TO_TIME2 := DINT_TO_TIME(UDINT_TO_DINT(IN));

END_FUNCTION

FUNCTION_BLOCK T_PLC_MS_block
	VAR_OUTPUT
		T_PLC_MS :	UDINT;
	END_VAR

	VAR_EXTERNAL
		PLC_TICKS_PER_SEC :	INT;
		PLC_SYS_TICK_CNT :	DINT;
	END_VAR

	VAR
		debug :	BOOL;(*Debug-Mode ON / OFF*)
		N :	INT;(*Debug-Faktor*)
		Offset :	UDINT;(*Debug-Offset*)
		temp :	DWORD := DWORD#1;(*Debug-Offset*)
		mode :	BOOL;(*modus*)
		faktor :	UDINT;(*Systemtakt-Faktor*)
		init :	BOOL;
		v_plc_ticks_per_sec :	UDINT;
		base :	UDINT := UDINT#1000;
	END_VAR

	IF init = FALSE THEN
		v_plc_ticks_per_sec := INT_TO_UDINT(PLC_TICKS_PER_SEC);
		IF v_plc_ticks_per_sec = UDINT#1024 THEN
			faktor := UDINT#1;
			mode := FALSE;
		ELSIF v_plc_ticks_per_sec > UDINT#0 THEN
			IF v_plc_ticks_per_sec <= base THEN
				faktor := base / v_plc_ticks_per_sec;
				mode := FALSE;
			ELSE
				faktor := v_plc_ticks_per_sec / base;
				mode := TRUE;
			END_IF;
		ELSE
			faktor := UDINT#1;
		END_IF;
		init := TRUE;
	END_IF;

	IF mode THEN
		T_PLC_MS := DINT_TO_UDINT(PLC_SYS_TICK_CNT) / faktor;
	ELSE
		T_PLC_MS := DINT_TO_UDINT(PLC_SYS_TICK_CNT) * faktor;
	END_IF;

	IF debug THEN
		T_PLC_MS := (DWORD_TO_UDINT(SHL(UDINT_TO_DWORD(T_PLC_MS),N) OR SHL(temp,N)) - UDINT#1) + Offset;
	END_IF;

END_FUNCTION_BLOCK

FUNCTION_BLOCK PULSE_T_Block

	VAR_INPUT
		IN :	BOOL;
		T1 :	TIME;
		T2 :	TIME;
		RST :	BOOL;
	END_VAR

	VAR_OUTPUT
		Q :	BOOL;
	END_VAR

	VAR
		init :	BOOL;
		last :	TIME;
		tx :	TIME;
		edge :	BOOL;
		T_PLC_MS :	T_PLC_MS_Block;
	END_VAR

	T_PLC_MS();
	tx:= UDINT_TO_TIME(T_PLC_MS.T_PLC_MS);

	IF NOT init THEN
		init := TRUE;
		last := tx;
	ELSIF RST THEN
		Q := FALSE;
	ELSIF IN AND NOT edge AND NOT Q THEN
		last := tx;
		Q := TRUE;
	ELSIF NOT IN AND edge AND ((tx - last) > T1) THEN
		Q := FALSE;
	ELSIF (tx - last) >= T2 THEN
		Q := FALSE;
	END_IF;

	edge := IN;

END_FUNCTION_BLOCK

PROGRAM program0
	VAR
		IN :	BOOL;
		T1 :	TIME;
		T2 :	TIME;
		RST :	BOOL;
		Q :	BOOL;

		func_block : PULSE_T_Block;
	END_VAR
	func_block.IN := IN;
	func_block.T1 := T1;
	func_block.T2 := T2 ;
	func_block.RST := RST ;

	func_block();
	Q  := func_block.Q;
END_PROGRAM

CONFIGURATION Config0
	VAR_GLOBAL
		PLC_TICKS_PER_SEC :	INT;
		PLC_SYS_TICK_CNT :	DINT;
	END_VAR
  	RESOURCE Res0 ON PLC
    	TASK task0(INTERVAL := T#20ms,PRIORITY := 0);
    	PROGRAM instance0 WITH task0 : program0;
  	END_RESOURCE
END_CONFIGURATION

(* ---- PWM_DC.ST ---- *)
FUNCTION_BLOCK T_PLC_MS_block
	VAR_OUTPUT
		T_PLC_MS :	UDINT;
	END_VAR

	VAR_EXTERNAL
		PLC_TICKS_PER_SEC :	INT;
		PLC_SYS_TICK_CNT :	DINT;
	END_VAR

	VAR
		debug :	BOOL;(*Debug-Mode ON / OFF*)
		N :	INT;(*Debug-Faktor*)
		Offset :	UDINT;(*Debug-Offset*)
		temp :	DWORD := DWORD#1;(*Debug-Offset*)
		mode :	BOOL;(*modus*)
		faktor :	UDINT;(*Systemtakt-Faktor*)
		init :	BOOL;
		v_plc_ticks_per_sec :	UDINT;
		base :	UDINT := UDINT#1000;
	END_VAR

	IF init = FALSE THEN
		v_plc_ticks_per_sec := INT_TO_UDINT(PLC_TICKS_PER_SEC);
		IF v_plc_ticks_per_sec = UDINT#1024 THEN
			faktor := UDINT#1;
			mode := FALSE;
		ELSIF v_plc_ticks_per_sec > UDINT#0 THEN
			IF v_plc_ticks_per_sec <= base THEN
				faktor := base / v_plc_ticks_per_sec;
				mode := FALSE;
			ELSE
				faktor := v_plc_ticks_per_sec / base;
				mode := TRUE;
			END_IF;
		ELSE
			faktor := UDINT#1;
		END_IF;
		init := TRUE;
	END_IF;

	IF mode THEN
		T_PLC_MS := DINT_TO_UDINT(PLC_SYS_TICK_CNT) / faktor;
	ELSE
		T_PLC_MS := DINT_TO_UDINT(PLC_SYS_TICK_CNT) * faktor;
	END_IF;

	IF debug THEN
		T_PLC_MS := (DWORD_TO_UDINT(SHL(UDINT_TO_DWORD(T_PLC_MS),N) OR SHL(temp,N)) - UDINT#1) + Offset;
	END_IF;

END_FUNCTION_BLOCK

FUNCTION_BLOCK CLK_PRG
	VAR_INPUT
		PT :	TIME := T#10ms;
	END_VAR

	VAR_OUTPUT
		Q :	BOOL;
	END_VAR

	VAR
		init :	BOOL := FALSE;
		last :	TIME;
		tx :	TIME;
		T_PLC_MS :	T_PLC_MS_block;
	END_VAR

	T_PLC_MS();
	tx:= UDINT_TO_TIME(T_PLC_MS.T_PLC_MS);

	IF NOT init THEN
		init := TRUE;
		last := tx - pt;
	END_IF;

	Q := tx - last >= pt;
	IF Q THEN last := tx; END_IF;
END_FUNCTION_BLOCK

FUNCTION _REAL_TO_UDINT:UDINT
  VAR_INPUT
    X :	REAL;
  END_VAR

  IF REAL_TO_UDINT(0.5) = UDINT#1 THEN
    _REAL_TO_UDINT := REAL_TO_UDINT(x);
  ELSIF X > 0.0 THEN
    _REAL_TO_UDINT := REAL_TO_UDINT(x+0.5);
  ELSIF X < 0.0 THEN
    _REAL_TO_UDINT := REAL_TO_UDINT(x-0.5);
  ELSE
    _REAL_TO_UDINT := UDINT#0;
  END_IF;
END_FUNCTION

FUNCTION REAL_TO_TIME2:TIME
	VAR_INPUT
		IN :	REAL;
	END_VAR

	REAL_TO_TIME2 := DINT_TO_TIME(UDINT_TO_DINT(_REAL_TO_UDINT(IN)));
END_FUNCTION

FUNCTION_BLOCK TP_X
	VAR_INPUT
		IN :	BOOL;
		PT :	TIME;
	END_VAR

	VAR_OUTPUT
		Q :	BOOL;
		ET :	TIME;
	END_VAR

	VAR
		edge :	BOOL;
		start :	TIME;
		tx :	TIME;
		T_PLC_MS :	T_PLC_MS_block;
	END_VAR

	T_PLC_MS();
	tx := UDINT_TO_TIME(T_PLC_MS.T_PLC_MS);

	IF IN AND NOT edge THEN
		start := tx;
		Q := PT > t#0ms;
	ELSIF Q THEN
		ET := tx - start;
		IF ET >= PT THEN
			Q := FALSE;
			ET := t#0ms;
		END_IF;
	END_IF;
	edge := IN;

END_FUNCTION_BLOCK

FUNCTION_BLOCK PWM_DC
	VAR_INPUT
		F :	REAL;
		DC :	REAL;
	END_VAR

	VAR_OUTPUT
		Q :	BOOL;
	END_VAR

	VAR
		clk :	CLK_Prg;
		pulse :	TP_X;
		tmp :	REAL;
	END_VAR

	IF F > 0.0 THEN
		tmp := 1000.0/F;
		CLK(PT := REAL_TO_TIME2(tmp));
		Pulse(in := clk.Q, pt := REAL_TO_TIME2(tmp*DC));
		Q := pulse.Q;
	END_IF;
END_FUNCTION_BLOCK

PROGRAM program0
  VAR
	F  :	REAL;
	DC :	REAL;

	Q :	BOOL;

	func_block : PWM_DC;
  END_VAR
	func_block.F     :=F     ;
	func_block.DC    :=DC    ;
	func_block();
	Q := func_block.Q;
END_PROGRAM

CONFIGURATION Config0
	VAR_GLOBAL
		PLC_TICKS_PER_SEC :	INT;
		PLC_SYS_TICK_CNT :	DINT;
	END_VAR

  RESOURCE Res0 ON PLC
    TASK task0(INTERVAL := T#20ms,PRIORITY := 0);
    PROGRAM instance0 WITH task0 : program0;
  END_RESOURCE
END_CONFIGURATION

(* ---- R2_ABS.ST ---- *)
TYPE REAL2 :

	STRUCT
		R1 : REAL;
		RX : REAL;
	END_STRUCT;

END_TYPE

FUNCTION_BLOCK R2_ABS_Block

	VAR_INPUT
		X :	REAL2;
	END_VAR

	VAR_OUTPUT
		R2_ABS :	REAL2;
	END_VAR

	IF X.RX >= 0.0 THEN
		R2_ABS.RX := X.RX;
		R2_ABS.R1 := X.R1;
	ELSE
		R2_ABS.RX := -X.RX;
		R2_ABS.R1 := -X.R1;
	END_IF;

END_FUNCTION_BLOCK

PROGRAM program0

	VAR
		X :	REAL2;

        R2_ABS :	REAL2;
		func_block : R2_ABS_Block;
	END_VAR
	func_block.X := X;
	func_block();
	R2_ABS := func_block.R2_ABS;

END_PROGRAM

CONFIGURATION Config0

	RESOURCE Res0 ON PLC
		TASK task0(INTERVAL := T#20ms,PRIORITY := 0);
		PROGRAM instance0 WITH task0 : program0;
	END_RESOURCE

END_CONFIGURATION

(* ---- R2_ADD.ST ---- *)
TYPE REAL2 :

	STRUCT
		R1 : REAL;
		RX : REAL;
	END_STRUCT;

END_TYPE

FUNCTION_BLOCK R2_ADD_Block

	VAR_INPUT
		X :	REAL2;
		Y :	REAL;
	END_VAR

	VAR_OUTPUT
		R2_ADD :	REAL2;
	END_VAR

	VAR
		temp :	REAL;
	END_VAR

	temp := X.RX;
	R2_ADD.RX := Y + X.R1 + X.RX;
	R2_ADD.R1 := temp - R2_ADD.RX + Y + X.R1;

END_FUNCTION_BLOCK

PROGRAM program0

	VAR
		X :	REAL2;
		Y :	REAL;

        R2_ADD :	REAL2;
		func_block : R2_ADD_Block;
	END_VAR
	func_block.X := X;
	func_block.Y := Y;
	func_block();
	R2_ADD := func_block.R2_ADD;

END_PROGRAM

CONFIGURATION Config0

	RESOURCE Res0 ON PLC
		TASK task0(INTERVAL := T#20ms,PRIORITY := 0);
		PROGRAM instance0 WITH task0 : program0;
	END_RESOURCE

END_CONFIGURATION

(* ---- R2_ADD2.ST ---- *)
TYPE REAL2 :

	STRUCT
		R1 : REAL;
		RX : REAL;
	END_STRUCT;

END_TYPE

FUNCTION_BLOCK R2_ADD2_Block

	VAR_INPUT
		X :	REAL2;
		Y :	REAL2;
	END_VAR

	VAR_OUTPUT
		R2_ADD2 :	REAL2;
	END_VAR

	R2_ADD2.R1 := X.R1 + Y.R1;
	R2_ADD2.RX := X.RX + Y.RX;

END_FUNCTION_BLOCK

PROGRAM program0

	VAR
		X :	REAL2;
		Y :	REAL2;

        R2_ADD2 :	REAL2;
		func_block : R2_ADD2_Block;
	END_VAR
	func_block.X := X;
	func_block.Y := Y;
	func_block();
	R2_ADD2 := func_block.R2_ADD2;

END_PROGRAM

CONFIGURATION Config0

	RESOURCE Res0 ON PLC
		TASK task0(INTERVAL := T#20ms,PRIORITY := 0);
		PROGRAM instance0 WITH task0 : program0;
	END_RESOURCE

END_CONFIGURATION

(* ---- R2_DIV.ST ---- *)
TYPE REAL2 :

	STRUCT
		R1 : REAL;
		RX : REAL;
	END_STRUCT;

END_TYPE

FUNCTION_BLOCK R2_DIV_Block

	VAR_INPUT
		X :	REAL2;
		Y :	REAL;
	END_VAR

	VAR_OUTPUT
		R2_DIV :	REAL2;
	END_VAR

	R2_DIV.RX := X.RX / Y;
	R2_DIV.R1 := X.R1 / Y;

END_FUNCTION_BLOCK

PROGRAM program0

	VAR
		X :	REAL2;
		Y :	REAL;

        R2_DIV :	REAL2;
		func_block : R2_DIV_Block;
	END_VAR
	func_block.X := X;
	func_block.Y := Y;
	func_block();
	R2_DIV := func_block.R2_DIV;

END_PROGRAM

CONFIGURATION Config0

	RESOURCE Res0 ON PLC
		TASK task0(INTERVAL := T#20ms,PRIORITY := 0);
		PROGRAM instance0 WITH task0 : program0;
	END_RESOURCE

END_CONFIGURATION

(* ---- R2_MUL.ST ---- *)
TYPE REAL2 :

	STRUCT
		R1 : REAL;
		RX : REAL;
	END_STRUCT;

END_TYPE

FUNCTION_BLOCK R2_MUL_Block

	VAR_INPUT
		X :	REAL2;
		Y :	REAL;
	END_VAR

	VAR_OUTPUT
		R2_MUL :	REAL2;
	END_VAR

	R2_MUL.RX := X.RX * Y;
	R2_MUL.R1 := X.R1 * Y;

END_FUNCTION_BLOCK

PROGRAM program0

	VAR
		X :	REAL2;
		Y :	REAL;

        R2_MUL :	REAL2;
		func_block : R2_MUL_Block;
	END_VAR
	func_block.X := X;
	func_block.Y := Y;
	func_block();
	R2_MUL := func_block.R2_MUL;

	END_PROGRAM

CONFIGURATION Config0

	RESOURCE Res0 ON PLC
		TASK task0(INTERVAL := T#20ms,PRIORITY := 0);
		PROGRAM instance0 WITH task0 : program0;
	END_RESOURCE

END_CONFIGURATION

(* ---- R2_SET.ST ---- *)
TYPE REAL2 :

	STRUCT
		R1 : REAL;
		RX : REAL;
	END_STRUCT;

END_TYPE

FUNCTION_BLOCK R2_SET_Block

	VAR_INPUT
		X :	REAL;
	END_VAR

	VAR_OUTPUT
		R2_SET :	REAL2;
	END_VAR

	R2_SET.RX := X;
	R2_SET.R1 := 0.0;

END_FUNCTION_BLOCK

PROGRAM program0

	VAR
		X :	REAL;

        R2_SET :	REAL2;
		func_block : R2_SET_Block;
	END_VAR
	func_block.X := X;
	func_block();
	R2_SET := func_block.R2_SET;

	END_PROGRAM

CONFIGURATION Config0

	RESOURCE Res0 ON PLC
		TASK task0(INTERVAL := T#20ms,PRIORITY := 0);
		PROGRAM instance0 WITH task0 : program0;
	END_RESOURCE

END_CONFIGURATION

(* ---- RDM.ST ---- *)
FUNCTION D_TRUNC : DINT
  VAR_INPUT
    x : REAL;
  END_VAR

  D_TRUNC := REAL_TO_DINT(X);
  IF X > 0.0 THEN
  	IF DINT_TO_REAL(D_TRUNC) > X THEN D_TRUNC := D_TRUNC - DINT#1; END_IF;
  ELSE
  	IF DINT_TO_REAL(D_TRUNC) < X THEN D_TRUNC := D_TRUNC + DINT#1; END_IF;
  END_IF;
END_FUNCTION

FUNCTION BIT_COUNT:INT

	VAR_INPUT
		IN :	DWORD;
	END_VAR

	VAR
		in_temp :	DWORD;
	END_VAR

	in_temp := IN;
	WHILE in_temp > DWORD#0 DO
		IF (in_temp AND DWORD#16#00000001) > DWORD#0 THEN Bit_Count := Bit_Count +1; END_IF;
		in_temp := SHR(in_temp,1);
	END_WHILE;

END_FUNCTION

FUNCTION FRACT:REAL
	VAR_INPUT
		X :	REAL;
	END_VAR

	IF ABS(x) < 2.0E9 THEN
		FRACT := x - DINT_TO_REAL(D_TRUNC(x));
	ELSE
		FRACT := 0.0;
	END_IF;

END_FUNCTION

FUNCTION_BLOCK T_PLC_MS_block
	VAR_OUTPUT
		T_PLC_MS :	UDINT;
	END_VAR

	VAR_EXTERNAL
		PLC_TICKS_PER_SEC :	INT;
		PLC_SYS_TICK_CNT :	DINT;
	END_VAR

	VAR
		debug :	BOOL;(*Debug-Mode ON / OFF*)
		N :	INT;(*Debug-Faktor*)
		Offset :	UDINT;(*Debug-Offset*)
		temp :	DWORD := DWORD#1;(*Debug-Offset*)
		mode :	BOOL;(*modus*)
		faktor :	UDINT;(*Systemtakt-Faktor*)
		init :	BOOL;
		v_plc_ticks_per_sec :	UDINT;
		base :	UDINT := UDINT#1000;
	END_VAR

	IF init = FALSE THEN
		v_plc_ticks_per_sec := INT_TO_UDINT(PLC_TICKS_PER_SEC);
		IF v_plc_ticks_per_sec = UDINT#1024 THEN
			faktor := UDINT#1;
			mode := FALSE;
		ELSIF v_plc_ticks_per_sec > UDINT#0 THEN
			IF v_plc_ticks_per_sec <= base THEN
				faktor := base / v_plc_ticks_per_sec;
				mode := FALSE;
			ELSE
				faktor := v_plc_ticks_per_sec / base;
				mode := TRUE;
			END_IF;
		ELSE
			faktor := UDINT#1;
		END_IF;
		init := TRUE;
	END_IF;

	IF mode THEN
		T_PLC_MS := DINT_TO_UDINT(PLC_SYS_TICK_CNT) / faktor;
	ELSE
		T_PLC_MS := DINT_TO_UDINT(PLC_SYS_TICK_CNT) * faktor;
	END_IF;

	IF debug THEN
		T_PLC_MS := (DWORD_TO_UDINT(SHL(UDINT_TO_DWORD(T_PLC_MS),N) OR SHL(temp,N)) - UDINT#1) + Offset;
	END_IF;

END_FUNCTION_BLOCK

FUNCTION BIT_LOAD_DW:DWORD

	VAR_INPUT
		IN :	DWORD;
		VAL :	BOOL;
		POS :	INT;
	END_VAR

	IF val THEN
		BIT_LOAD_DW := in OR SHL(DWORD#1,pos);
	ELSE
		BIT_LOAD_DW := in AND (NOT SHL(DWORD#1,pos));
	END_IF;

END_FUNCTION

FUNCTION BIT_OF_DWORD : BOOL
  VAR_INPUT
    IN : DWORD;
    N : INT;
  END_VAR

  BIT_OF_DWORD := (SHR(in,N) AND 16#00000001) > 0;
  (* from OSCAT library; www.oscat.de  *)
END_FUNCTION

FUNCTION _INT_TO_UDINT:UDINT
	VAR_INPUT
		IN :	INT;
	END_VAR

	_INT_TO_UDINT := DINT_TO_UDINT(INT_TO_DINT(IN));
END_FUNCTION

FUNCTION _DWORD_TO_REAL:REAL
	VAR_INPUT
		IN :	DWORD;
	END_VAR

	_DWORD_TO_REAL := UDINT_TO_REAL(DWORD_TO_UDINT(IN));

END_FUNCTION

FUNCTION_BLOCK RDM_block
	VAR_INPUT
		LAST :	REAL;
	END_VAR
	VAR_OUTPUT
		RDM :	REAL;
	END_VAR
	VAR
		T_PLC_MS :	T_PLC_MS_block;
		tn :	DWORD;
		tc :	INT;
	END_VAR
	T_PLC_MS();
	tn := UDINT_TO_DWORD(T_PLC_MS.T_PLC_MS);
	tc := Bit_Count(tn);

	tn:=BIT_LOAD_DW(tn,BIT_OF_DWORD(tn,2),31); (* tn.31 := tn.2; *)
	tn:=BIT_LOAD_DW(tn,BIT_OF_DWORD(tn,5),30); (* tn.30 := tn.5; *)
	tn:=BIT_LOAD_DW(tn,BIT_OF_DWORD(tn,4),29); (* tn.29 := tn.4; *)
	tn:=BIT_LOAD_DW(tn,BIT_OF_DWORD(tn,1),28); (* tn.28 := tn.1; *)
	tn:=BIT_LOAD_DW(tn,BIT_OF_DWORD(tn,0),27); (* tn.27 := tn.0; *)
	tn:=BIT_LOAD_DW(tn,BIT_OF_DWORD(tn,7),26); (* tn.26 := tn.7; *)
	tn:=BIT_LOAD_DW(tn,BIT_OF_DWORD(tn,6),25); (* tn.25 := tn.6; *)
	tn:=BIT_LOAD_DW(tn,BIT_OF_DWORD(tn,3),24); (* tn.24 := tn.3; *)

	tn := ROL(tn,Bit_Count(tn)) OR DWORD#16#80000001;
	tn := UDINT_TO_DWORD(DWORD_TO_UDINT(tn) MOD UDINT#71474513 + _INT_TO_UDINT(tc) + UDINT#77);
	RDM := fract(_DWORD_TO_REAL(tn) / 10000000.0 * (2.71828182845904523536028747135266249 - LIMIT_REAL(0.0,last,1.0)));
END_FUNCTION_BLOCK

PROGRAM program0
	VAR
	    LocalVar : REAL;
		LocalOUT  : REAL;
		func_block : RDM_block;
  	END_VAR
	func_block.LAST := LocalVar;
	func_block();
	LocalOUT := func_block.RDM;
END_PROGRAM

CONFIGURATION Config0
	VAR_GLOBAL
		PLC_TICKS_PER_SEC :	INT;
		PLC_SYS_TICK_CNT :	DINT;
	END_VAR

  	RESOURCE Res0 ON PLC
    	TASK task0(INTERVAL := T#20ms,PRIORITY := 0);
    	PROGRAM instance0 WITH task0 : program0;
  	END_RESOURCE
END_CONFIGURATION

(* ---- RDM2.ST ---- *)
FUNCTION _REAL_TO_DWORD: DWORD
	VAR_INPUT
		X :	REAL;
	END_VAR

	IF REAL_TO_DWORD(0.5) = DWORD#1 THEN
		_REAL_TO_DWORD := REAL_TO_DWORD(x);
	ELSIF X > 0.0 THEN
		_REAL_TO_DWORD := REAL_TO_DWORD(x+0.5);
	ELSIF X < 0.0 THEN
		_REAL_TO_DWORD := REAL_TO_DWORD(x-0.5);
	ELSE
		_REAL_TO_DWORD := DWORD#0;
	END_IF;
END_FUNCTION

FUNCTION _DWORD_TO_REAL:REAL
	VAR_INPUT
		IN :	DWORD;
	END_VAR

	_DWORD_TO_REAL := UDINT_TO_REAL(DWORD_TO_UDINT(IN));

END_FUNCTION

FUNCTION _INT_TO_UDINT:UDINT
	VAR_INPUT
		IN :	INT;
	END_VAR

	_INT_TO_UDINT := DINT_TO_UDINT(INT_TO_DINT(IN));
END_FUNCTION

FUNCTION D_TRUNC : DINT
	VAR_INPUT
		x : REAL;
	END_VAR

	D_TRUNC := REAL_TO_DINT(X);
	IF X > 0.0 THEN
		IF DINT_TO_REAL(D_TRUNC) > X THEN D_TRUNC := D_TRUNC - DINT#1; END_IF;
	ELSE
		IF DINT_TO_REAL(D_TRUNC) < X THEN D_TRUNC := D_TRUNC + DINT#1; END_IF;
	END_IF;
END_FUNCTION

FUNCTION FRACT:REAL
	VAR_INPUT
		X :	REAL;
	END_VAR

	IF ABS(x) < 2.0E9 THEN
		FRACT := x - DINT_TO_REAL(D_TRUNC(x));
	ELSE
		FRACT := 0.0;
	END_IF;
END_FUNCTION

FUNCTION BIT_LOAD_DW:DWORD

	VAR_INPUT
		IN :	DWORD;
		VAL :	BOOL;
		POS :	INT;
	END_VAR

	IF val THEN
		BIT_LOAD_DW := in OR SHL(DWORD#1,pos);
	ELSE
		BIT_LOAD_DW := in AND (NOT SHL(DWORD#1,pos));
	END_IF;
END_FUNCTION

FUNCTION BIT_OF_DWORD : BOOL
	VAR_INPUT
		IN : DWORD;
		N : INT;
	END_VAR

	BIT_OF_DWORD := (SHR(in,N) AND 16#00000001) > 0;
END_FUNCTION

FUNCTION BIT_COUNT:INT
	VAR_INPUT
		IN :	DWORD;
	END_VAR

	VAR
		in_temp :	DWORD;
	END_VAR

	in_temp := IN;
	WHILE in_temp > DWORD#0 DO
		IF (in_temp AND DWORD#16#00000001) > DWORD#0 THEN Bit_Count := Bit_Count +1; END_IF;
		in_temp := SHR(in_temp,1);
	END_WHILE;
END_FUNCTION

FUNCTION_BLOCK T_PLC_MS_Block
	VAR_OUTPUT
		T_PLC_MS :	UDINT;
	END_VAR

	VAR_EXTERNAL
		PLC_TICKS_PER_SEC :	INT;
		PLC_SYS_TICK_CNT :	DINT;
	END_VAR

	VAR
		debug :	BOOL;(*Debug-Mode ON / OFF*)
		N :	INT;(*Debug-Faktor*)
		Offset :	UDINT;(*Debug-Offset*)
		temp :	DWORD := DWORD#1;(*Debug-Offset*)
		mode :	BOOL;(*modus*)
		faktor :	UDINT;(*Systemtakt-Faktor*)
		init :	BOOL;
		v_plc_ticks_per_sec :	UDINT;
		base :	UDINT := UDINT#1000;
	END_VAR

	IF init = FALSE THEN
		v_plc_ticks_per_sec := INT_TO_UDINT(PLC_TICKS_PER_SEC);
		IF v_plc_ticks_per_sec = UDINT#1024 THEN
			faktor := UDINT#1;
			mode := FALSE;
		ELSIF v_plc_ticks_per_sec > UDINT#0 THEN
			IF v_plc_ticks_per_sec <= base THEN
				faktor := base / v_plc_ticks_per_sec;
				mode := FALSE;
			ELSE
				faktor := v_plc_ticks_per_sec / base;
				mode := TRUE;
			END_IF;
		ELSE
			faktor := UDINT#1;
		END_IF;
		init := TRUE;
	END_IF;

	IF mode THEN
		T_PLC_MS := DINT_TO_UDINT(PLC_SYS_TICK_CNT) / faktor;
	ELSE
		T_PLC_MS := DINT_TO_UDINT(PLC_SYS_TICK_CNT) * faktor;
	END_IF;

	IF debug THEN
		T_PLC_MS := (DWORD_TO_UDINT(SHL(UDINT_TO_DWORD(T_PLC_MS),N) OR SHL(temp,N)) - UDINT#1) + Offset;
	END_IF;
END_FUNCTION_BLOCK

FUNCTION_BLOCK RDM_Block
	VAR_INPUT
		LAST :	REAL;
	END_VAR
	VAR_OUTPUT
		RDM :	REAL;
	END_VAR
	VAR
		T_PLC_MS :	T_PLC_MS_Block;
		tn :	DWORD;
		tc :	INT;
	END_VAR
	T_PLC_MS();
	tn := UDINT_TO_DWORD(T_PLC_MS.T_PLC_MS);
	tc := Bit_Count(tn);

	tn:=BIT_LOAD_DW(tn,BIT_OF_DWORD(tn,2),31); (* tn.31 := tn.2; *)
	tn:=BIT_LOAD_DW(tn,BIT_OF_DWORD(tn,5),30); (* tn.30 := tn.5; *)
	tn:=BIT_LOAD_DW(tn,BIT_OF_DWORD(tn,4),29); (* tn.29 := tn.4; *)
	tn:=BIT_LOAD_DW(tn,BIT_OF_DWORD(tn,1),28); (* tn.28 := tn.1; *)
	tn:=BIT_LOAD_DW(tn,BIT_OF_DWORD(tn,0),27); (* tn.27 := tn.0; *)
	tn:=BIT_LOAD_DW(tn,BIT_OF_DWORD(tn,7),26); (* tn.26 := tn.7; *)
	tn:=BIT_LOAD_DW(tn,BIT_OF_DWORD(tn,6),25); (* tn.25 := tn.6; *)
	tn:=BIT_LOAD_DW(tn,BIT_OF_DWORD(tn,3),24); (* tn.24 := tn.3; *)

	tn := ROL(tn,Bit_Count(tn)) OR DWORD#16#80000001;
	tn := UDINT_TO_DWORD(DWORD_TO_UDINT(tn) MOD UDINT#71474513 + _INT_TO_UDINT(tc) + UDINT#77);
	RDM := fract(_DWORD_TO_REAL(tn) / 10000000.0 * (2.71828182845904523536028747135266249 - LIMIT_REAL(0.0,last,1.0)));
END_FUNCTION_BLOCK

FUNCTION_BLOCK RDM2_Block
	VAR_INPUT
		LAST :	INT;
		LOW :	INT;
		HIGH :	INT;
	END_VAR

	VAR_OUTPUT
		RDM2 :	INT;
	END_VAR

	VAR
		rdm :	RDM_Block;
	END_VAR

	rdm(last:=fract(INT_TO_REAL(last) * 3.14159265358979323846264338327950288));
	RDM2 := TRUNC(rdm.RDM * INT_TO_REAL(high - low + 1)) + low;

END_FUNCTION_BLOCK

PROGRAM program0

	VAR
		LAST :	INT;
		LOW :	INT;
		HIGH :	INT;

        RDM2 :	INT;
		func_block : RDM2_Block;
	END_VAR
		func_block.LAST := LAST;
		func_block.LOW := LOW;
		func_block.HIGH := HIGH;
		func_block();
		RDM2 := func_block.RDM2;

END_PROGRAM

CONFIGURATION Config0

	VAR_GLOBAL
		PLC_TICKS_PER_SEC :	INT;
		PLC_SYS_TICK_CNT :	DINT;
	END_VAR

	RESOURCE Res0 ON PLC
		TASK task0(INTERVAL := T#20ms,PRIORITY := 0);
		PROGRAM instance0 WITH task0 : program0;
	END_RESOURCE

END_CONFIGURATION

(* ---- RDMDW.ST ---- *)
FUNCTION _REAL_TO_DWORD: DWORD
	VAR_INPUT
		X :	REAL;
	END_VAR

	IF REAL_TO_DWORD(0.5) = DWORD#1 THEN
		_REAL_TO_DWORD := REAL_TO_DWORD(x);
	ELSIF X > 0.0 THEN
		_REAL_TO_DWORD := REAL_TO_DWORD(x+0.5);
	ELSIF X < 0.0 THEN
		_REAL_TO_DWORD := REAL_TO_DWORD(x-0.5);
	ELSE
		_REAL_TO_DWORD := DWORD#0;
	END_IF;
END_FUNCTION

FUNCTION _DWORD_TO_REAL:REAL
	VAR_INPUT
		IN :	DWORD;
	END_VAR

	_DWORD_TO_REAL := UDINT_TO_REAL(DWORD_TO_UDINT(IN));

END_FUNCTION

FUNCTION _INT_TO_UDINT:UDINT
	VAR_INPUT
		IN :	INT;
	END_VAR

	_INT_TO_UDINT := DINT_TO_UDINT(INT_TO_DINT(IN));
END_FUNCTION

FUNCTION D_TRUNC : DINT
	VAR_INPUT
		x : REAL;
	END_VAR

	D_TRUNC := REAL_TO_DINT(X);
	IF X > 0.0 THEN
		IF DINT_TO_REAL(D_TRUNC) > X THEN D_TRUNC := D_TRUNC - DINT#1; END_IF;
	ELSE
		IF DINT_TO_REAL(D_TRUNC) < X THEN D_TRUNC := D_TRUNC + DINT#1; END_IF;
	END_IF;
END_FUNCTION

FUNCTION FRACT:REAL
	VAR_INPUT
		X :	REAL;
	END_VAR

	IF ABS(x) < 2.0E9 THEN
		FRACT := x - DINT_TO_REAL(D_TRUNC(x));
	ELSE
		FRACT := 0.0;
	END_IF;
END_FUNCTION

FUNCTION BIT_LOAD_DW:DWORD

	VAR_INPUT
		IN :	DWORD;
		VAL :	BOOL;
		POS :	INT;
	END_VAR

	IF val THEN
		BIT_LOAD_DW := in OR SHL(DWORD#1,pos);
	ELSE
		BIT_LOAD_DW := in AND (NOT SHL(DWORD#1,pos));
	END_IF;
END_FUNCTION

FUNCTION BIT_OF_DWORD : BOOL
	VAR_INPUT
		IN : DWORD;
		N : INT;
	END_VAR

	BIT_OF_DWORD := (SHR(in,N) AND 16#00000001) > 0;
END_FUNCTION

FUNCTION BIT_COUNT:INT
	VAR_INPUT
		IN :	DWORD;
	END_VAR

	VAR
		in_temp :	DWORD;
	END_VAR

	in_temp := IN;
	WHILE in_temp > DWORD#0 DO
		IF (in_temp AND DWORD#16#00000001) > DWORD#0 THEN Bit_Count := Bit_Count +1; END_IF;
		in_temp := SHR(in_temp,1);
	END_WHILE;
END_FUNCTION

FUNCTION_BLOCK T_PLC_MS_Block
	VAR_OUTPUT
		T_PLC_MS :	UDINT;
	END_VAR

	VAR_EXTERNAL
		PLC_TICKS_PER_SEC :	INT;
		PLC_SYS_TICK_CNT :	DINT;
	END_VAR

	VAR
		debug :	BOOL;(*Debug-Mode ON / OFF*)
		N :	INT;(*Debug-Faktor*)
		Offset :	UDINT;(*Debug-Offset*)
		temp :	DWORD := DWORD#1;(*Debug-Offset*)
		mode :	BOOL;(*modus*)
		faktor :	UDINT;(*Systemtakt-Faktor*)
		init :	BOOL;
		v_plc_ticks_per_sec :	UDINT;
		base :	UDINT := UDINT#1000;
	END_VAR

	IF init = FALSE THEN
		v_plc_ticks_per_sec := INT_TO_UDINT(PLC_TICKS_PER_SEC);
		IF v_plc_ticks_per_sec = UDINT#1024 THEN
			faktor := UDINT#1;
			mode := FALSE;
		ELSIF v_plc_ticks_per_sec > UDINT#0 THEN
			IF v_plc_ticks_per_sec <= base THEN
				faktor := base / v_plc_ticks_per_sec;
				mode := FALSE;
			ELSE
				faktor := v_plc_ticks_per_sec / base;
				mode := TRUE;
			END_IF;
		ELSE
			faktor := UDINT#1;
		END_IF;
		init := TRUE;
	END_IF;

	IF mode THEN
		T_PLC_MS := DINT_TO_UDINT(PLC_SYS_TICK_CNT) / faktor;
	ELSE
		T_PLC_MS := DINT_TO_UDINT(PLC_SYS_TICK_CNT) * faktor;
	END_IF;

	IF debug THEN
		T_PLC_MS := (DWORD_TO_UDINT(SHL(UDINT_TO_DWORD(T_PLC_MS),N) OR SHL(temp,N)) - UDINT#1) + Offset;
	END_IF;
END_FUNCTION_BLOCK

FUNCTION_BLOCK RDM_Block
	VAR_INPUT
		LAST :	REAL;
	END_VAR
	VAR_OUTPUT
		RDM :	REAL;
	END_VAR
	VAR
		T_PLC_MS :	T_PLC_MS_Block;
		tn :	DWORD;
		tc :	INT;
	END_VAR
	T_PLC_MS();
	tn := UDINT_TO_DWORD(T_PLC_MS.T_PLC_MS);
	tc := Bit_Count(tn);

	tn:=BIT_LOAD_DW(tn,BIT_OF_DWORD(tn,2),31); (* tn.31 := tn.2; *)
	tn:=BIT_LOAD_DW(tn,BIT_OF_DWORD(tn,5),30); (* tn.30 := tn.5; *)
	tn:=BIT_LOAD_DW(tn,BIT_OF_DWORD(tn,4),29); (* tn.29 := tn.4; *)
	tn:=BIT_LOAD_DW(tn,BIT_OF_DWORD(tn,1),28); (* tn.28 := tn.1; *)
	tn:=BIT_LOAD_DW(tn,BIT_OF_DWORD(tn,0),27); (* tn.27 := tn.0; *)
	tn:=BIT_LOAD_DW(tn,BIT_OF_DWORD(tn,7),26); (* tn.26 := tn.7; *)
	tn:=BIT_LOAD_DW(tn,BIT_OF_DWORD(tn,6),25); (* tn.25 := tn.6; *)
	tn:=BIT_LOAD_DW(tn,BIT_OF_DWORD(tn,3),24); (* tn.24 := tn.3; *)

	tn := ROL(tn,Bit_Count(tn)) OR DWORD#16#80000001;
	tn := UDINT_TO_DWORD(DWORD_TO_UDINT(tn) MOD UDINT#71474513 + _INT_TO_UDINT(tc) + UDINT#77);
	RDM := fract(_DWORD_TO_REAL(tn) / 10000000.0 * (2.71828182845904523536028747135266249 - LIMIT_REAL(0.0,last,1.0)));
END_FUNCTION_BLOCK

FUNCTION_BLOCK RDMDW_Block

	VAR_INPUT
		LAST :	DWORD;
	END_VAR

	VAR_OUTPUT
		RDMDW :	DWORD;
	END_VAR

	VAR
		RX :	REAL;
		M :	REAL;
		rdm :	RDM_Block;
	END_VAR

	M := INT_TO_REAL(BIT_COUNT(last));
	rdm(last:=FRACT(M*3.14159265358979323846264338327950288));
	RX:=rdm.RDM;
	RDMDW := SHL(_REAL_TO_DWORD(rx*65535.0),16);

	rdm(last:=FRACT(M*2.71828182845904523536028747135266249));
	RX:=rdm.RDM;
	RDMDW := RDMDW OR (_REAL_TO_DWORD(rx*65535.0) AND DWORD#16#0000FFFF);

END_FUNCTION_BLOCK

PROGRAM program0

	VAR
		LAST :	DWORD;

        RDMDW :	DWORD;
		func_block : RDMDW_Block;
	END_VAR
		func_block.LAST := LAST;
		func_block();
		RDMDW := func_block.RDMDW;

END_PROGRAM

CONFIGURATION Config0

	VAR_GLOBAL
		PLC_TICKS_PER_SEC :	INT;
		PLC_SYS_TICK_CNT :	DINT;
	END_VAR

	RESOURCE Res0 ON PLC
		TASK task0(INTERVAL := T#20ms,PRIORITY := 0);
		PROGRAM instance0 WITH task0 : program0;
	END_RESOURCE

END_CONFIGURATION

(* ---- REAL_TO_FRAC.ST ---- *)
TYPE oscat_FRACTION :
	STRUCT
		NUMERATOR : INT;
		DENOMINATOR : INT;
	END_STRUCT;
END_TYPE

FUNCTION_BLOCK REAL_TO_FRAC_Block

	VAR_INPUT
		X :	REAL;
		N :	INT;
	END_VAR

	VAR_OUTPUT
		REAL_TO_FRAC :	oscat_FRACTION;
	END_VAR

	VAR
		temp :	DINT;
		sign :	BOOL;
		X_gerundet :	DINT;
		X_ohne_Nachkomma :	REAL;
		Numerator :	DINT := 1;
		Denominator :	DINT := 0;
		Numerator_old :	DINT := 0;
		Denominator_old :	DINT := 1;
	END_VAR

	IF X < 0.0 THEN
		sign := TRUE;								(* Vorzeichen merken *)
		X := ABS(X);								(* Absolutwert berechnen *)
	END_IF;

	REPEAT
		X_gerundet := REAL_TO_DINT(X);

		temp := numerator * X_gerundet + numerator_old;		(* Zaehler um Vorkammawert erweitern *)
		numerator_old := numerator;							(* Zaehler der letzten Berechnung speichern *)
		numerator := temp;									(* Zaehler dieser Berechnung speichern *)

		temp := denominator * X_gerundet + denominator_old;	(* Nenner um Vorkammawert erweitern *)
		denominator_old := denominator;						(* Nenner der letzten Berechnung speichern *)
		denominator := temp;								(* Nenner dieser Berechnung speichern *)

		X_ohne_Nachkomma := DINT_TO_REAL(X_gerundet);
		IF X = X_ohne_Nachkomma THEN						(* Bruch geht ohne Rest auf *)
			IF ABS(denominator) <= INT_TO_DINT(N) THEN		(* kein Rundungsfehler *)
				numerator_old := numerator;					(* Numerator_old wird von Funktion zur�ckgegeben *)
				denominator_old := denominator;				(* Denominator_old wird von Funktion zur�ckgegeben *)
			END_IF;
			EXIT;											(* keine weitere Berechnung notwendig *)
		ELSE
			X := 1.0 / (X - X_ohne_Nachkomma);				(* Kehrwert vom Rest -> Neuer Bruch *)
		END_IF;

	UNTIL
		( ABS(Denominator) > INT_TO_DINT(N))
	END_REPEAT;

	IF sign THEN
		REAL_TO_FRAC.NUMERATOR := -1 * ABS(DINT_TO_INT(numerator_old));
	ELSE
		REAL_TO_FRAC.NUMERATOR :=  ABS(DINT_TO_INT(numerator_old));
	END_IF;

	REAL_TO_FRAC.DENOMINATOR := ABS(DINT_TO_INT(denominator_old));

END_FUNCTION_BLOCK

PROGRAM program0

	VAR
		X :	REAL;
		N :	INT;

        REAL_TO_FRAC :	oscat_FRACTION;
		func_block : REAL_TO_FRAC_Block;
	END_VAR
		func_block.X := X;
		func_block.N := N;
		func_block();
		REAL_TO_FRAC := func_block.REAL_TO_FRAC;

END_PROGRAM

CONFIGURATION Config0

	RESOURCE Res0 ON PLC
		TASK task0(INTERVAL := T#20ms,PRIORITY := 0);
		PROGRAM instance0 WITH task0 : program0;
	END_RESOURCE

END_CONFIGURATION

(* ---- REAL_TO_STRF.ST ---- *)
FUNCTION EXP10 : REAL

	VAR_INPUT
		x : REAL;
	END_VAR

	exp10 := EXP(X * 2.30258509299405);

END_FUNCTION

FUNCTION _REAL_TO_DINT:DINT
	VAR_INPUT
		X :	REAL;
	END_VAR

	IF REAL_TO_DINT(0.5) = DINT#1 THEN
		_REAL_TO_DINT := REAL_TO_DINT(x);
		RETURN;
	END_IF;

	IF X > 0.0 THEN
		_REAL_TO_DINT := REAL_TO_DINT(x+0.5);
	ELSIF X < 0.0 THEN
		_REAL_TO_DINT := REAL_TO_DINT(x-0.5);
	ELSE
		_REAL_TO_DINT := DINT#0;
	END_IF;
END_FUNCTION

FUNCTION_BLOCK REAL_TO_STRF_Block

	VAR_INPUT
		IN :	REAL;
		N :	INT;
		D :	STRING;
	END_VAR

	VAR_OUTPUT
		REAL_TO_STRF :	STRING;
	END_VAR

	VAR
		st_tmp : STRING;
		i :	INT;
	END_VAR

	N := LIMIT(0,N,7);
	REAL_TO_STRF := DINT_TO_STRING(_REAL_TO_DINT(ABS(in) * EXP10(INT_TO_REAL(N))));
	FOR i := LEN(REAL_TO_STRF) TO N DO
		st_tmp := REAL_TO_STRF;
		REAL_TO_STRF := CONCAT('0', st_tmp);
	END_FOR;
	IF n > 0 THEN REAL_TO_STRF := INSERT(REAL_TO_STRF, D, LEN(REAL_TO_STRF) - N); END_IF;
	IF in < 0.0 THEN st_tmp := REAL_TO_STRF; REAL_TO_STRF := CONCAT('-', st_tmp); END_IF;

END_FUNCTION_BLOCK

PROGRAM program0

	VAR
		IN :	REAL;
		N :	INT;
		D :	STRING;

        REAL_TO_STRF :	STRING;
		func_block : REAL_TO_STRF_Block;
	END_VAR
		func_block.IN := IN;
		func_block.N := N;
		func_block.D := D;
		func_block();
		REAL_TO_STRF := func_block.REAL_TO_STRF;

END_PROGRAM

CONFIGURATION Config0

	RESOURCE Res0 ON PLC
		TASK task0(INTERVAL := T#20ms,PRIORITY := 0);
		PROGRAM instance0 WITH task0 : program0;
	END_RESOURCE

END_CONFIGURATION

(* ---- REPLACE_ALL.ST ---- *)
FUNCTION_BLOCK FINDP_Block

	VAR_INPUT
		STR :	STRING;
		SRC :	STRING;
		POS :	INT;
	END_VAR

	VAR_OUTPUT
		FINDP :	INT;
	END_VAR

	VAR
		i :	INT;
		ls :	INT;
		lx :	INT;
		stp :	INT;
		st_tmp :	STRING;
	END_VAR

	ls := LEN(str);
	lx := LEN(src);
	IF ls < lx OR lx = 0 THEN RETURN; END_IF;
	stp := ls - lx + 1;
	FOR i := MAX(pos,1) TO stp DO
		st_tmp := MID(str,lx,i);
		IF EQ_STRING(st_tmp,src) THEN
			FINDP := i;
			RETURN;
		END_IF;
	END_FOR;
	FINDP := 0;

END_FUNCTION_BLOCK

FUNCTION_BLOCK REPLACE_ALL_Block

	VAR_INPUT
		STR :	STRING;
		SRC :	STRING;
		REP :	STRING;
	END_VAR

	VAR_OUTPUT
		REPLACE_ALL :	STRING;
	END_VAR

	VAR
		pos :	INT;
		lp :	INT;
		lx :	INT;
		FINDP :	FINDP_Block;
		st_tmp :	STRING;
	END_VAR

	REPLACE_ALL := str;
	lx := LEN(src);
	lp := LEN(rep);

	FINDP.str := REPLACE_ALL;
	FINDP.src := src;
	FINDP.pos := 1;
	FINDP();
	pos := FINDP.FINDP;

	WHILE pos > 0 DO
		st_tmp := REPLACE_ALL;
		REPLACE_ALL := REPLACE(st_tmp,rep,lx,pos);

		FINDP.str := REPLACE_ALL;
		FINDP.src := src;
		FINDP.pos := pos + lp;
		FINDP();
		pos := FINDP.FINDP;

	END_WHILE;

END_FUNCTION_BLOCK

PROGRAM program0

	VAR
		STR :	STRING;
		SRC :	STRING;
		REP :	STRING;

        REPLACE_ALL :	STRING;
		func_block : REPLACE_ALL_Block;
	END_VAR
		func_block.STR := STR;
		func_block.SRC := SRC;
		func_block.REP := REP;
		func_block();
		REPLACE_ALL := func_block.REPLACE_ALL;

END_PROGRAM

CONFIGURATION Config0

	RESOURCE Res0 ON PLC
		TASK task0(INTERVAL := T#20ms,PRIORITY := 0);
		PROGRAM instance0 WITH task0 : program0;
	END_RESOURCE

END_CONFIGURATION
